(* IEC 61131-3 sources: ConveyorControl-with-PLC/4E_Gruppe1_Graf_Projekt1/Class/SdiasManager (part 3) *)

//**********************************************************************************************************************************************************
    CMD_GET_HARDWARE_DIAGNOSIS:
      //Returns module info
      ret_code := ERROR;
      pResult^.aData[0]$t_HWCGetHardwareDiagnosisOut.retcode := _HWC_RETVAL_ERROR;

      pStr_HWTRequested := pPara^.aPara[0]$t_HWCGetHardwareDiagnosisIn.pStr_HardewareTreeEntry;

      if pStr_HWTRequested &
         ( ((pStr_HWTRequested  + pPara^.aPara[0]$t_HWCGetHardwareTreeEntryIn.us_current_index  - 1)^$USINT) = HWT_ESCAPE_SDIAS ) then

        tmpplace := (pStr_HWTRequested+pPara^.aPara[0]$t_HWCGetHardwareDiagnosisIn.us_current_index)^$USINT;

        //Check if pointer is valid
        if ModuleObjInfo[tmpplace].pThis then
          ret_code := ModuleObjInfo[tmpplace].pThis^.NewInst(pPara,pResult);
        else
          pResult^.aData[0]$t_HWCGetHardwareDiagnosisOut.retcode := _HWC_RETVAL_ERROR_SDIAS_MODULE_NOT_FOUND;
        end_if;
      end_if;

//**********************************************************************************************************************************************************
    CMD_GET_HARDWARE_TREE_ENTRY:
      //Returns module info
      ret_code := ERROR;
      pResult^.aData[0]$t_HWCGetHardwareTreeEntryOut.retcode := _HWC_RETVAL_ERROR;

      pStr_HWTreeEntry := pPara^.aPara[0]$t_HWCGetHardwareTreeEntryIn.pStr_LastHardewareTreeEntry;

      //First HWT Path
      if pStr_HWTreeEntry = nil then
        if ModuleObjInfo[0].pThis then

          ret_code := ModuleObjInfo[0].pThis^.NewInst(pPara,pResult);
        else
          pResult^.aData[0]$t_HWCGetHardwareTreeEntryOut.retcode := _HWC_RETVAL_ERROR_SDIAS_MODULE_NOT_FOUND;
        end_if;

      //search next module
      elsif ( ((pStr_HWTreeEntry  + pPara^.aPara[0]$t_HWCGetHardwareTreeEntryIn.us_current_index  - 1)^$USINT) = HWT_ESCAPE_SDIAS ) then

        // Check last modul again incase it was an extension module
        usNextPlace := (pStr_HWTreeEntry  + pPara^.aPara[0]$t_HWCGetHardwareTreeEntryIn.us_current_index)^$USINT;
        if ModuleObjInfo[usNextPlace].pThis then

          ret_code := ModuleObjInfo[usNextPlace].pThis^.NewInst(pPara,pResult);
        else
          ret_code := READY;
          pResult^.aData$t_HWCGetHardwareTreeEntryOut.retcode := _HWC_RETVAL_OK_END_OF_LIST;
          return;
        end_if;

        // Module was found, return next one
        if ret_code = READY &
           (pResult^.aData$t_HWCGetHardwareTreeEntryOut.retcode = _HWC_RETVAL_OK_MODULE_FOUND |
            pResult^.aData$t_HWCGetHardwareTreeEntryOut.retcode = _HWC_RETVAL_OK_END_OF_LIST) then

          usNextPlace += 1;
          if ModuleObjInfo[usNextPlace].pThis then

            ret_code := ModuleObjInfo[usNextPlace].pThis^.NewInst(pPara,pResult);
          else
            ret_code := READY;
            pResult^.aData$t_HWCGetHardwareTreeEntryOut.retcode := _HWC_RETVAL_OK_END_OF_LIST;
          end_if;

        end_if;

      end_if;

//**********************************************************************************************************************************************************

//*****************************************************************************
//** COMMANDS FROM SDIAS MODULES                                             **
//*****************************************************************************

    // port number is always stored in pPara^.aPara[MAXCMDPARA-1]
//**********************************************************************************************************************************************************
		SDIAS_CMD_ADD_RD_ACCESS:
      if AddAccess(_Read, pPara^.aPara[0]$^SdiasBase, pPara^.aPara[1]$UDINT, pPara^.aPara[2], pPara^.aPara[3]$HINT, pPara^.aPara[4]$UINT, pPara^.aPara[5]$pVoid, pPara^.aPara[6]$pVoid, pPara^.aPara[7]$pVoid, pPara^.aPara[8]$^UDINT, pPara^.aPara[9]$UDINT, pPara^.aPara[10]$BOOL) = FALSE then
        ret_code := ERROR;
      end_if;

//**********************************************************************************************************************************************************
    SDIAS_CMD_ADD_WR_ACCESS:
      if AddAccess(_Write, pPara^.aPara[0]$^SdiasBase, pPara^.aPara[1]$UDINT, pPara^.aPara[2], pPara^.aPara[3]$HINT, pPara^.aPara[4]$UINT, pPara^.aPara[5]$pVoid, pPara^.aPara[6]$pVoid, pPara^.aPara[7]$pVoid, pPara^.aPara[8]$^UDINT, pPara^.aPara[9]$UDINT, pPara^.aPara[10]$BOOL) = FALSE then
        ret_code := ERROR;
      end_if;

//**********************************************************************************************************************************************************
		SDIAS_CMD_ADD_DYN_RD_ACCESS:
      if AddAccess(_ReadDynamic, pPara^.aPara[0]$^SdiasBase, pPara^.aPara[1]$UDINT, pPara^.aPara[2], pPara^.aPara[3]$HINT, pPara^.aPara[4]$UINT, pPara^.aPara[5]$pVoid, pPara^.aPara[6]$pVoid, pPara^.aPara[7]$pVoid, pPara^.aPara[8]$^UDINT, pPara^.aPara[9]$UDINT, pPara^.aPara[10]$BOOL) = FALSE then
        ret_code := ERROR;
      end_if;

//**********************************************************************************************************************************************************
    SDIAS_CMD_ADD_DYN_WR_ACCESS:
      if AddAccess(_WriteDynamic, pPara^.aPara[0]$^SdiasBase, pPara^.aPara[1]$UDINT, pPara^.aPara[2], pPara^.aPara[3]$HINT, pPara^.aPara[4]$UINT, pPara^.aPara[5]$pVoid, pPara^.aPara[6]$pVoid, pPara^.aPara[7]$pVoid, pPara^.aPara[8]$^UDINT, pPara^.aPara[9]$UDINT, pPara^.aPara[10]$BOOL) = FALSE then
        ret_code := ERROR;
      end_if;

//**********************************************************************************************************************************************************
    SDIAS_CMD_CHANGE_DYN_ACCESS:
      if ChangeDynAccess(AccessHandle:=pPara^.aPara[0]$UDINT, NewOffset:=pPara^.aPara[1]$UDINT, NewLength:=pPara^.aPara[2]$UDINT) = FALSE then
        ret_code := ERROR;
      end_if;

//**********************************************************************************************************************************************************
    SDIAS_CMD_SDO_SEND_REQUEST:

      if pPara^.aPara[1]$t_SDIAS_SDO_Cmd = SDIAS_SDO_CMD_SPI_READ & FirmwareVersion < SDIAS_SDO_SPI_FIRMWARE_VERSION_AVAILABLE then
        LogError(e_msg:="SdiasManager::ClassState::NewInst: SPI Read failed, Update FirmwareVersion of SDIAS Manager");
        ret_code := ERROR;
        return;
      end_if;

      if AddSDOReq(pCmdSvr:=pPara^.aPara[0]$^SvrChCmd, Command:=pPara^.aPara[1]$t_SDIAS_SDO_Cmd, Place:=pPara^.aPara[2]$USINT, CmdLength:=pPara^.aPara[3]$USINT, pReqBuf:=pPara^.aPara[4]$^USINT) <> SDIAS_OK then
        ret_code := ERROR;
      end_if;

//**********************************************************************************************************************************************************
    SDIAS_CMD_CHANGE_LED_STATE:
      // get byte position ouf of place (place 0-3 in byte 0, 4-7 in byte 1,...)
      ByteNr := pPara^.aPara[1]$USINT SHR 2;
      PosInByte := (pPara^.aPara[1]$USINT AND 2#11) SHL 1;
      AppliLEDStates[ByteNr] := (AppliLEDStates[ByteNr] AND NOT(2#11 SHL PosInByte)) OR (pPara^.aPara[2]$USINT SHL PosInByte);
      b_NewLEDStates := TRUE;

//**********************************************************************************************************************************************************
    SDIAS_CMD_DA_RD_ACCESS:
      // not implemented yet
      ret_code := ERROR;

//      DaWriteBuffer.ReadLength  := pPara^.aPara[1]$USINT;
//      DaWriteBuffer.ReadOffset  := pPara^.aPara[0]$HINT;
//      DaWriteBuffer.WriteLength := 0;
//      DaWriteBuffer.WriteOffset := 0;
//
//      DaWriteBuffer.TriggerUnit := sizeof(t_DAWrPayloadFrame) - sizeof(t_DAWrPayloadFrame.Data); // no data sent on reading
//
//      DAPara.ud_AddOffset := DaWriteOffset;
//      DAPara.ud_length    := DaWriteBuffer.TriggerUnit;
//      DAPara.p_ud_data    := (#DaWriteBuffer)$^UDINT;
//
//      tempCmd.uiCmd := _BUS_IF_WR_DA;
//      tempCmd.aPara[0] := (#DAPara)$DINT;
//      ToBusInterface.NewInst(pPara:=#tempCmd, pResult:=#_result);
//
//      if _result.aData[4]$t_BusIFRetvalErrorcode <> _BUS_IF_RETVAL_OK then
//        LogError("(SdiasManager::ClassState::NewInst) Direct access write on VARAN failed as part of the SDIAS direct access read!");
//        ret_code := ERROR;
//      else
//        DAPara.ud_AddOffset := DaReadOffset;
//        DAPara.ud_length    := DaWriteBuffer.ReadLength + sizeof(t_SDIAS_StateByte);
//        DAPara.p_ud_data    := (#DaReadBuffer)$^UDINT;
//
//        tempCmd.uiCmd := _BUS_IF_RD_DA;
//        tempCmd.aPara[0] := (#DAPara)$DINT;
//        ToBusInterface.NewInst(pPara:=#tempCmd, pResult:=#_result);
//
//        if _result.aData[4]$t_BusIFRetvalErrorcode <> _BUS_IF_RETVAL_OK then
//          LogError("(SdiasManager::ClassState::NewInst) Direct access read on VARAN failed as part of the SDIAS direct access read!");
//          ret_code := ERROR;
//        else
//          // copy the read data to the user memory
//          _memcpy(ptr1:=pPara^.aPara[2]$^USINT, ptr2:=#DaReadBuffer.Data, cntr:=DaWriteBuffer.ReadLength);
//        end_if;
//      end_if;

//**********************************************************************************************************************************************************
    SDIAS_CMD_DA_WR_ACCESS:
      // not implemented yet
      ret_code := ERROR;

//      DaWriteBuffer.ReadLength  := 0;
//      DaWriteBuffer.ReadOffset  := 0;
//      DaWriteBuffer.WriteLength := pPara^.aPara[1]$USINT;
//      DaWriteBuffer.WriteOffset := pPara^.aPara[0]$HINT;
//
//      DaWriteBuffer.TriggerUnit := sizeof(t_DAWrPayloadFrame) - sizeof(t_DAWrPayloadFrame.Data) + DaWriteBuffer.WriteLength; // no data sent on reading
//
//      // copy the write data from the user memory
//      _memcpy(ptr1:=#DaWriteBuffer.Data, ptr2:=pPara^.aPara[2]$^USINT, cntr:=DaWriteBuffer.WriteLength);
//
//      DAPara.ud_AddOffset := DaWriteOffset;
//      DAPara.ud_length    := DaWriteBuffer.TriggerUnit;
//      DAPara.p_ud_data    := (#DaWriteBuffer)$^UDINT;
//
//      tempCmd.uiCmd := _BUS_IF_WR_DA;
//      tempCmd.aPara[0] := (#DAPara)$DINT;
//      ToBusInterface.NewInst(pPara:=#tempCmd, pResult:=#_result);
//
//      if _result.aData[4]$t_BusIFRetvalErrorcode <> _BUS_IF_RETVAL_OK then
//        LogError("(SdiasManager::ClassState::NewInst) Direct access write on VARAN failed as part of the SDIAS direct access write!");
//        ret_code := ERROR;
//      else
//        DAPara.ud_AddOffset := DaReadOffset;
//        DAPara.ud_length    := sizeof(t_SDIAS_StateByte);
//        DAPara.p_ud_data    := (#DaReadBuffer)$^UDINT;
//
//        tempCmd.uiCmd := _BUS_IF_RD_DA;
//        tempCmd.aPara[0] := (#DAPara)$DINT;
//        ToBusInterface.NewInst(pPara:=#tempCmd, pResult:=#_result);
//
//        if _result.aData[4]$t_BusIFRetvalErrorcode <> _BUS_IF_RETVAL_OK then
//          LogError("(SdiasManager::ClassState::NewInst) Direct access read on VARAN failed as part of the SDIAS direct access write!");
//          ret_code := ERROR;
//        end_if;
//      end_if;

//**********************************************************************************************************************************************************
    SDIAS_CMD_REQUIRED_ERROR:
      SetRequiredError(pTargetThis:=pPara^.aPara[0]$^SdiasBase, Place:=pPara^.aPara[1]$UDINT);

//**********************************************************************************************************************************************************
    SDIAS_CMD_INIT_STATE_LOGIN:
      Place := pPara^.aPara[1]$UDINT;
      if (Place <= SDIAS_MAX_PLACE_NR) & pPara^.aPara[0] then
        ModuleObjInfo[Place].pInitState       := pPara^.aPara[0]$^t_e_VaranErrors;
        ModuleObjInfo[Place].pThis            := pPara^.aPara[2]$^SdiasBase;

        // get task settings
        ModuleObjInfo[Place].bPreScan         := (pPara^.aPara[3] AND SDIAS_TASK_MASK_RT_PRE ) <> 0;
        ModuleObjInfo[Place].bPostScan        := (pPara^.aPara[3] AND SDIAS_TASK_MASK_RT_POST) <> 0;
        ModuleObjInfo[Place].bCyclic          := (pPara^.aPara[3] AND SDIAS_TASK_MASK_CY     ) <> 0;

        // get access structure
        ModuleObjInfo[Place].pDefaultAccesses := pPara^.aPara[4]$^t_SDIAS_DefaultAccesses;

        // required info
        ModuleObjInfo[Place].Required         := pPara^.aPara[5];

        if ModuleObjInfo[Place].Required & (b_SDIASModulesRequired = FALSE) then
          b_SDIASModulesRequired := TRUE;
          // if any access is required => the businterface is also required
          tempCmd.uiCmd := _BUS_IF_SET_REQUIRED;
          ToBusInterface.NewInst(pPara:=#tempCmd, pResult:=#_result);
          if _result.aData[0]$t_BusIFRetvalErrorcode <> _BUS_IF_RETVAL_OK then
            LogError("(SdiasManager::ClassState::NewInst) Failed to set the BusInterface to required");
          end_if;
        end_if;

        // remember the highest place to save time in module scanning operations like calling the realtime methods
        if (Place > MaxPlace) | (MaxPlace = SDIAS_PLACE_NO_MODULE_ADDED_SO_FAR) then
          MaxPlace := Place;
        end_if;
      else
        ret_code := ERROR;
      end_if;

//**********************************************************************************************************************************************************
    SDIAS_CMD_GET_HW_PATH:
      // forward it to bus interface
      pPara^.uiCmd := _BUS_IF_GET_HW_PATH;
      ret_code := ToBusInterface.NewInst(pPara, pResult);

//**********************************************************************************************************************************************************
    SDIAS_CMD_INSTALL_CYCLIC_TASK:
      ModuleObjInfo[pPara^.aPara[0]].bCyclic := TRUE;

//**********************************************************************************************************************************************************
    SDIAS_CMD_GET_CONNECTION_TYPE:
      pResult^.uiLng := sizeof(t_SDIAS_ConnectionType);
      pResult^.aData[0]$t_SDIAS_ConnectionType := ConnectionType;

//**********************************************************************************************************************************************************
    SDIAS_CMD_CREATE_MUTEX:
      // forward it to bus interface
      pPara^.uiCmd := _BUS_IF_CREATE_MUTEX;
      ret_code := ToBusInterface.NewInst(pPara, pResult);

//**********************************************************************************************************************************************************
    SDIAS_CMD_IS_VARAN_AVAILABLE:
      // forward it to bus interface
      pPara^.uiCmd := _BUS_IF_IS_VARAN_AVAILABLE;
      ret_code := ToBusInterface.NewInst(pPara, pResult);

//**********************************************************************************************************************************************************
    SDIAS_CMD_ADD_DEVICE_ID:
    //add valid ids to list
    for i:= 0 to 9 do
      //Check if no id is stored or if id is already stored in list.
      if aValidDeviceIDs[i] = 0 | aValidDeviceIDs[i] = pPara^.aPara[0]$UDINT then
        aValidDeviceIDs[i] := pPara^.aPara[0]$UDINT;
        exit;
      end_if;
    end_for;

//**********************************************************************************************************************************************************

//*****************************************************************************
//** COMMANDS FORWARDED BY SDIAS BUS INTERFACE                               **
//*****************************************************************************

//**********************************************************************************************************************************************************
    _BUS_IF_ADD_MOVE_DO:
      // correct the parameters, because the calling class doesn't have the information
      pDataADDMove                        := (pPara^.aPara[0])$^t_AddMoveDOCfg;

      pDataADDMove^.ud_handle_source      := ISOReadDO.AccessHandle;
      pDataADDMove^.ud_addressoff_source  := pDataADDMove^.p_sourcedata$UDINT - ISOReadDO.pData$UDINT;

      // if we have the DPRAM address extra => recalculate the address
      if ISOReadDO.pDataDPRAM then
        pDataADDMove^.p_sourcedata := ISOReadDO.pDataDPRAM + pDataADDMove^.ud_addressoff_source;
      end_if;

      pDataADDMove^.ud_handle_dest        := ISOWriteDO.AccessHandle;
      pDataADDMove^.ud_addressoff_dest    := pDataADDMove^.p_destdata$UDINT - ISOWriteDO.pData$UDINT;

      // if we have the DPRAM address extra => recalculate the address
      if ISOWriteDO.pDataDPRAM then
        pDataADDMove^.p_destdata := ISOWriteDO.pDataDPRAM + pDataADDMove^.ud_addressoff_dest;
      end_if;

      // forward it to bus interface
      ret_code := ToBusInterface.NewInst(pPara, pResult);

//**********************************************************************************************************************************************************
    _BUS_IF_UPDATE_MOVE_DO:
      // forward it to bus interface
      ret_code := ToBusInterface.NewInst(pPara, pResult);

//**********************************************************************************************************************************************************
    _BUS_IF_GET_ACCESS_INFO:
      // check if we got a valid pointer (local memory)
      if pPara^.aPara[0] then
        // return the access info
        pResult^.uiLng := sizeof(t_AccessInfoRet);
        pAccessInfo := (#pResult^.aData[0])$^t_AccessInfoRet;

        pAccessInfo^.ud_handle     := ISOReadDO.AccessHandle;
        pAccessInfo^.ud_addressoff := pPara^.aPara[0]$UDINT - ISOReadDO.pData$UDINT;

        // if we have the DPRAM address extra => recalculate the address
        if ISOReadDO.pDataDPRAM then
          pAccessInfo^.p_dataDPRAM := ISOReadDO.pDataDPRAM + pAccessInfo^.ud_addressoff;
        end_if;
      end_if;

//**********************************************************************************************************************************************************

//*****************************************************************************
//** COMMANDS FROM BUS INTERFACE                                             **
//*****************************************************************************

//**********************************************************************************************************************************************************
    _BUS_IF_HWCONNECT :
      // device has been connected. if there is no bus ready signal or we're in the init (no bus ready in init if module is already connected) => do the connect-stuff here
      ConnectEvent();
      pResult^.aData[0] := _BUS_IF_RETVAL_OK;

//**********************************************************************************************************************************************************
    _BUS_IF_HWSUB_BUS_READY :
      // we wait for the device bitmap to match => do nothing here
      pResult^.aData[0] := _BUS_IF_RETVAL_OK;

//**********************************************************************************************************************************************************
    _BUS_IF_HWDISCONNECT :
      // device has been disconnected
      DisconnectEvent();
      pResult^.aData[0] := _BUS_IF_RETVAL_OK;

//**********************************************************************************************************************************************************
    _BUS_IF_HWINTERRUPT :
      // error at device which may lead to a disconnect or replace the disconnect callback
      InterruptEvent();
      pResult^.aData[0] := _BUS_IF_RETVAL_OK;

//**********************************************************************************************************************************************************
    _BUS_IF_CHECK_DEVICE_ID :
      // check for correct device id

      pResult^.aData[0] := (DeviceID = pPara^.aPara[0]$UDINT);
      if pResult^.aData[0] = false then
        for i:= 0 to 9 do
          //Id found?
          if aValidDeviceIDs[i] = pPara^.aPara[0]$UDINT then
            pResult^.aData[0] := TRUE;
            exit;
          end_if;
        end_for;
      end_if;

//**********************************************************************************************************************************************************
    _BUS_IF_GET_TASK_INFO:
      // we must fetch the task info before the image with the payload is copied to ensure correct data and correct error detection

      // on local SDIAS we have to fetch it from the OS
      if ConnectionType = SDIAS_CON_LOCAL_uC then
        if SDIAS_iGetNodePropertyIndexLen(hNodeHandle   := udNodeHandle
                                     , udIndex          := 1
                                     , udPropertyId     := SDM_PROP_TASK_INFO
                                     , udBufferLength   := sizeof(t_TaskInfoData) - sizeof(t_TaskInfoData.ErrorInfoFlags) - sizeof(t_TaskInfoData.Reserved)
                                     , pucBuf           := (#RdTaskInfo.Handshake)$^USINT
                                     ) <> SDIAS_OK then
          CyclicMsgMarker.PostIt.GetRdInfoFailed := TRUE;
        end_if;
        if SDIAS_iGetNodePropertyIndex(hNodeHandle      := udNodeHandle
                                     , udIndex          := 1
                                     , udPropertyId     := SDM_PROP_TASK_ERROR_INFO_FLAGS
                                     , pudPropertyValue := (#RdTaskInfo.ErrorInfoFlags)$^UDINT
                                     ) <> SDIAS_OK then
          CyclicMsgMarker.PostIt.GetRdInfoFailed := TRUE;
        end_if;

        if SDIAS_iGetNodePropertyIndexLen(hNodeHandle   := udNodeHandle
                                     , udIndex          := 2
                                     , udPropertyId     := SDM_PROP_TASK_INFO
                                     , udBufferLength   := sizeof(t_TaskInfoData) - sizeof(t_TaskInfoData.ErrorInfoFlags) - sizeof(t_TaskInfoData.Reserved)
                                     , pucBuf           := (#WrTaskInfo.Handshake)$^USINT
                                     ) <> SDIAS_OK then
          CyclicMsgMarker.PostIt.GetWrInfoFailed := TRUE;

        end_if;
        if SDIAS_iGetNodePropertyIndex(hNodeHandle      := udNodeHandle
                                     , udIndex          := 2
                                     , udPropertyId     := SDM_PROP_TASK_ERROR_INFO_FLAGS
                                     , pudPropertyValue := (#WrTaskInfo.ErrorInfoFlags)$^UDINT
                                     ) <> SDIAS_OK then
          CyclicMsgMarker.PostIt.GetWrInfoFailed := TRUE;
        end_if;
      end_if;

//**********************************************************************************************************************************************************
    _BUS_IF_POST_INIT_RT_READY:
      // if we got an error => return it
      if InitSSW = _ErrorOccured then
        ret_code := ERROR;

      // if we're not ready, return busy
      elsif RtSSW <> _Operational then
        ret_code := BUSY;
      end_if;

//**********************************************************************************************************************************************************
    _BUS_IF_CREATE_MUTEX,
    _BUS_IF_SET_REQUIRED_ERROR,
    _BUS_IF_GET_BUSCYCLE_TIME,
    _BUS_IF_GET_DEACTIVATED_STATE,
    _BUS_IF_GET_HW_PATH,
    _BUS_IF_IS_VARAN_AVAILABLE,
    _BUS_IF_SET_RUN_STATE,
    _BUS_IF_SET_REQUIRED:
      // forward it to bus interface
      ret_code := ToBusInterface.NewInst(pPara, pResult);
//**********************************************************************************************************************************************************

//*****************************************************************************
//** COMMANDS FROM SDIAS MANAGER ITSELF                                      **
//*****************************************************************************

//**********************************************************************************************************************************************************
		SDIAS_CMD_SDO_RESPONSE:
      ret_code := ReceiveSDOResponse(Command:=pPara^.aPara[0]$t_SDIAS_SDO_Cmd,
                                     Offset:=pPara^.aPara[1]$HINT,
                                     Length:=pPara^.aPara[2]$USINT,
                                     Result:=pPara^.aPara[3]$iprStates,
                                     pResponseBuffer:=pPara^.aPara[4]$^USINT,
                                     ResponseLength:=pPara^.aPara[5]$USINT
                                     );

//**********************************************************************************************************************************************************
  else
    // unknown command
    LogValue("(SdiasManager::ClassState::NewInst) Unknown command: 0x{0}", pPara^.uiCmd);
    ret_code := ERROR;
	END_CASE;

END_FUNCTION

FUNCTION SdiasManager::AddAccess
	VAR_INPUT
		AccessType 	: t_eAccessType;
		pThis 	: ^SdiasBase;
		Place 	: UDINT;
		Required 	: DINT;
		Offset 	: HINT;
		Length 	: UINT;
		ppData 	: pVoid;
		ppStateByte 	: pVoid;
		ppControlByte 	: pVoid;
		pAccessHandle 	: ^UDINT;
		WaitForAccessHandle 	: UDINT;
		bCtrlAcc0 	: BOOL;
	END_VAR
	VAR_OUTPUT
		Success 	: BOOL;
	END_VAR

  // check place
  if Place <= SDIAS_MAX_PLACE_NR then
    // check this pointer
    if pThis then
      // check other pointers as input parameters
      if ppData & ppStateByte & ppControlByte then
        // check offset and length for valid access
        if (Length > 0) & ((Offset + Length) <= SIZE_PER_SDIAS_CLIENT) then

          // remember the highest place to save time in module scanning operations like calling the realtime methods
          if (Place > MaxPlace) | (MaxPlace = SDIAS_PLACE_NO_MODULE_ADDED_SO_FAR) then
            MaxPlace := Place;
          end_if;

          // if it's a dynamic access on local SDIAS, check if the OS-Interface is available
          if ConnectionType = SDIAS_CON_LOCAL_uC then
            if ((AccessType = _ReadDynamic) | (AccessType = _WriteDynamic)) & (pSDIAS^.udVersion < SDIAS_CIL_VERSION_SUPPORTS_DYNAMIC_DO) then
              LogValue("(SdiasManager::AddAccess) Newer OS Version needed for dynamic accesses on local SDIAS. Access for module at place 0x{0} can't be created!", Place);
              ModuleObjInfo[Place].pInitState^ := _UnknownCommand;
              InitError := _UnknownCommand;
              Success := FALSE;
              return;
            end_if;
          end_if;

          // remember the access
          Success := AddAccessToList(AccessType           := AccessType,
                                     Place                := Place,
                                     Offset               := Offset,
                                     Length               := Length,
                                     ppData               := ppData,
                                     ppStateByte          := ppStateByte,
                                     ppControlByte        := ppControlByte,
                                     pAccessHandle        := pAccessHandle,
                                     WaitForAccessHandle  := WaitForAccessHandle,
                                     bCtrlAcc0            := bCtrlAcc0
                                     );

          // if adding failed classstate and initerrorstate are already set
          if Success = FALSE then
            LogValue("(SdiasManager::AddAccess) Failed to add Access for Module at Place 0x{0}", Place);
          end_if;
        else
          LogValue("(SdiasManager::AddAccess) Invalid access for module at place: 0x{0}. Check offset (0x{1}) and length (0x{2})!", Place, Offset, Length);
          ModuleObjInfo[Place].pInitState^ := _DOLAddressInvalid;
          InitError := _DOLAddressInvalid;
          Success := FALSE;
        end_if;
      else
        LogValue("(SdiasManager::AddAccess) Invalid pointer as input parameter for module at place: 0x{0}", Place);
        ModuleObjInfo[Place].pInitState^ := _MemoryFault;
        InitError := _MemoryFault;
        Success := FALSE;
      end_if;
    else
      LogValue("(SdiasManager::AddAccess) Invalid this pointer for module at place: 0x{0}", Place);
      ModuleObjInfo[Place].pInitState^ := _MemoryFault;
      InitError := _MemoryFault;
      Success := FALSE;
    end_if;
  else
    LogValue("(SdiasManager::AddAccess) Invalid Place number: 0x{0}. Maximum is 0x{1}", Place, SDIAS_MAX_PLACE_NR);
    if pThis then
      pThis^.ClassState := _InvalidDeviceAddress;
    end_if;
    InitError := _InvalidDeviceAddress;
    Success := FALSE;
  end_if;

  // if it was an access of a required module => required error
  if Required & (Success = FALSE) then
    SetRequiredError(pThis, Place);
  end_if;

END_FUNCTION

FUNCTION SdiasManager::ConnectEvent
  VAR
  	tempCmd         : CmdStruct;
    _result         : results;
    dataResetDO     : t_ResetDOCfg;
    Settings        : t_LoginSettings;
  END_VAR

  if b_PostInitFinished = FALSE then
    ConnectDuringPostInitCounter += 1;

    // don't reinit in postinit (ignore call from OS)
    if ConnectDuringPostInitCounter >= 2 then
      b_MultipleConnectInInit := TRUE;
      return;
    end_if;
  end_if;

  // install post init call back only if we're still in init (if we install it in init(), we may get called even the module is not connected)
  if us_Firstscan < 12 then
    tempCmd.uiCmd := _BUS_IF_WAIT_4_POST_INIT;
#pragma warning(disable: 74);
    Settings := 0;
#pragma warning(default: 74);
    Settings.Wait4DOCreation := MaxPlace <> SDIAS_PLACE_NO_MODULE_ADDED_SO_FAR;
    if Settings.Wait4DOCreation & (ConnectionType = SDIAS_CON_VIA_VARAN_uC) then
      Settings.Wait4MoveDOCreation := TRUE;
    end_if;
    Settings.Wait4SyncSend := TRUE;

    tempCmd.aPara[0] := Settings;
    ToBusInterface.NewInst(pPara:=#tempCmd, pResult:=#_result);

    if _result.aData[0]$t_BusIFRetvalErrorcode <> _BUS_IF_RETVAL_OK then
      LogError("(SdiasManager::ClassState::NewInst) Failed to install post init callback");
      InitError := _InvalidConfguration;
    end_if;
  else
    b_PostInitFinished := TRUE;
  end_if;

  if ConnectionType = SDIAS_CON_VIA_VARAN_uC then

    // reset data objects (calculate retry timeout)
    tempCmd.uiCmd     := _BUS_IF_RESET_DO;
    tempCmd.aPara[0]  := (#dataResetDO)$DINT;

    dataResetDO.Handle := ASYReadDO.Handle;

    ToBusInterface.NewInst(pPara:=#tempCmd, pResult:=#_result);
    if _result.aData[0]$t_BusIFRetvalErrorcode <> _BUS_IF_RETVAL_OK then
      LogError("(SdiasManager::ConnectEvent) Failed reset DO for the asynchronous read data");
    end_if;

    dataResetDO.Handle := ASYWriteDO.Handle;

    ToBusInterface.NewInst(pPara:=#tempCmd, pResult:=#_result);
    if _result.aData[0]$t_BusIFRetvalErrorcode <> _BUS_IF_RETVAL_OK then
      LogError("(SdiasManager::ConnectEvent) Failed reset DO for the asynchronous write data");
    end_if;
  end_if;

  // reset max durations as it marks the first run
  WriteTaskInfo.MaxDuration := 0;
  ReadTaskInfo.MaxDuration := 0;

  InitSSW := _StartInit;
  b_Ready4Rt := FALSE;
  RtSSW := _RtIdle;
  ClassState := _NotInitialized;
  Online := 1;

END_FUNCTION

FUNCTION SdiasManager::DisconnectEvent
  VAR
  	i : UDINT;
  END_VAR

  // if there is a required error, we would disguise it, if we call the disconnect interfaces
  if ClassState <> _RequiredError then

    // tell all the connected modules
    if MaxPlace <> SDIAS_PLACE_NO_MODULE_ADDED_SO_FAR then
      for i := 0 to MaxPlace do
        if ModuleObjInfo[i].pThis then
          ModuleObjInfo[i].pThis^.DisconnectEvent();
        end_if;
      end_for;
    end_if;

    ClassState := _NoHardware;

    FirmwareVersion := 0;
  end_if;

  Online := 0;

END_FUNCTION

FUNCTION SdiasManager::InterruptEvent

  // set only the state (we're in the interrupt and have to be fast)
  if b_IsRequired then
    ClassState := _HardwareRequiredIRQ;
  else
    ClassState := _HardwareNotRequiredIRQ;
  end_if;

  Online := 0;

END_FUNCTION

FUNCTION SdiasManager::SdiasManager
	VAR_OUTPUT
		ret_code 	: ConfStates;
	END_VAR
  VAR
    p_SSR			: ^LSL_SSR;
  END_VAR

  ClassState := _NotInitialized;

  //get pointer for logging function
	if ( OS_CILGET( "SSR", #p_SSR ) ) then
    p_KernelLog := NIL;
  else
    //Log function is available
		p_KernelLog := ( p_SSR^.KernelLog )$^DINT;
  end_if;

  //get pointer for sdias function
	if OS_CILGET( INTERFACE_SDIAS, #pSDIAS ) then
    LogError(e_msg:="(SdiasManager::SdiasManager) Failed to get SDIAS OS-Interface. A newer OS is necessary to use SDIAS");
  end_if;

  if (OS_CILGet("LSL_MULTITASK", #mt_api$void)) THEN
    LogError(e_msg:="(SdiasManager::SdiasManager) Failed to get MULTITASK OS-Interface for Mutex usage");
  end_if;

  MaxPlace := SDIAS_PLACE_NO_MODULE_ADDED_SO_FAR;

	ret_code := C_OK;

END_FUNCTION

FUNCTION VIRTUAL SdiasManager::LogError
	VAR_INPUT
		e_msg 	: ^CHAR;
	END_VAR
  VAR
    sz_name : ARRAY [ 0..255 ] OF CHAR;
  END_VAR

  _GetObjName( this, #sz_name[ 0 ] );

  MyTrace(pFormat:="ObjectName {0}: {1}", pTxt0:=(#sz_name[ 0 ])$^CHAR, pTxt1:= e_msg, pTxt2:=NIL);

END_FUNCTION

FUNCTION VIRTUAL SdiasManager::LogValue
	VAR_INPUT
		pString 	: ^CHAR;
		Value 	: UDINT;
		Value2 	: UDINT;(* := 16#FFFFFFFF *)
		Value3 	: UDINT;(* := 16#FFFFFFFF *)
	END_VAR
  VAR
    TempStr       : ARRAY [0..99] OF CHAR;
    TempStr2      : ARRAY [0..99] OF CHAR;
    TempStr3      : ARRAY [0..99] OF CHAR;
    TraceVal      : USINT;
    sz_name       : ARRAY [ 0..255 ] OF CHAR;
    TmpWithObjName: ARRAY [ 0..255 ] OF CHAR;
  END_VAR

  // number of values
  TraceVal := 1;

  _itoa(Value, #TempStr[0]);

  if pString <> NIL then
    _GetObjName( this, #sz_name[ 0 ] );
    _strcpy(dest:=#TmpWithObjName[0], src:="ObjectName ");
    _strcat(dest:=#TmpWithObjName[0], src:=#sz_name[0]);
    _strcat(dest:=#TmpWithObjName[0], src:=": ");
    _strcat(dest:=#TmpWithObjName[0], src:=pString);

    if Value2 <> 16#FFFFFFFF then
      _itoa(Value2, #TempStr2[0]);
      TraceVal += 1;
    end_if;

    if Value3 <> 16#FFFFFFFF then
      _itoa(Value3, #TempStr3[0]);
      TraceVal += 1;
    end_if;

    case TraceVal of
      1:MyTrace(pFormat:=#TmpWithObjName[0], pTxt0:=#TempStr[0], pTxt1:=NIL, pTxt2:=NIL);
      2:MyTrace(pFormat:=#TmpWithObjName[0], pTxt0:=#TempStr[0], pTxt1:=#TempStr2[0], pTxt2:=NIL);
      3:MyTrace(pFormat:=#TmpWithObjName[0], pTxt0:=#TempStr[0], pTxt1:=#TempStr2[0], pTxt2:=#TempStr3[0]);
    end_case;
  else
    MyTrace(pFormat:="<invalid string>", pTxt0:=NIL, pTxt1:=NIL, pTxt2:=NIL);
  end_if;

END_FUNCTION

FUNCTION VIRTUAL SdiasManager::MyTrace
	VAR_INPUT
		pFormat 	: ^CHAR;
		pTxt0 	: ^CHAR;
		pTxt1 	: ^CHAR;
		pTxt2 	: ^CHAR;
	END_VAR
  VAR
    nLen      : UDINT;
    pChr      : ^CHAR;
    nTxt      : UDINT;
    nRpl      : UDINT;
    pTxt      : ^CHAR;
    pText     : ^CHAR;
    FormText  : ARRAY [0 .. 255] OF CHAR;
  END_VAR

  // this method is a workaround for the TRACE message limitation problem

  pText := #FormText[0];

  _memset(dest:=#FormText[0], usByte:=0, cntr:=256); // to keep the zero termination

  _strncpy(pText, pFormat, 250);
  nLen  := _strlen(pText);
  pChr  := pText;

  WHILE nLen DO
    IF pChr^ = '{' THEN         // works for the first 10 replacement texts (single digit numbers)
      nTxt  := (pChr+1)^ - '0';
      CASE nTxt OF
        0:  pTxt  := pTxt0;
        1:  pTxt  := pTxt1;
        2:  pTxt  := pTxt2;
      ELSE
        pTxt  := "INV";
      END_CASE;
      nRpl  := _strlen(pTxt);
      if nLen - 3 + nRpl > 250 then
        pTxt := "LEN";  // replace the replacement text with "LEN" to see that we're out of length for this string
        nRpl := 3;
      end_if;
      _memmove(pChr + nRpl, pChr + 3, nLen);
      _memcpy(pChr, pTxt, nRpl);
      pChr  += nRpl;  // next character to parse is after the replacement text
      nLen  -= 3;     // the remaining length of the format string is decremented by 3
      if nLen > 250 then  // catch overrun of nLen
        nLen := 0;
      end_if;
    ELSE
      pChr  += 1;
      nLen  -= 1;
    END_IF;
  END_WHILE;

  TRACE(#FormText[0]);
  if ( p_KernelLog ) then
    OS_KERNELLOG0(#FormText[0]);
  end_if;

END_FUNCTION

FUNCTION SdiasManager::ChangeAsyRd
	VAR_INPUT
		Offset 	: HINT;
		Length 	: USINT;
		RunState 	: t_BusIFRunState;
		UsageType 	: t_AsyDOUsage;
	END_VAR
	VAR_OUTPUT
		Success 	: BOOL;
	END_VAR
  VAR
    dataUPDATEDO    : t_UpdateDOCfg;
  	tempCmd         : CmdStruct;
    _result         : results;
    dataSETRUNSTATE : t_SetRunStateCfg;
  END_VAR

  if (AsyReadUsage = _NotUsed) | (AsyReadUsage = UsageType) then

    // if length = zero we may just want to stop the DO
    if Length then
      ASYReadDO.Offset := Offset;
      ASYReadDO.Length := Length;

      dataUPDATEDO.Handle               := ASYReadDO.Handle;
      dataUPDATEDO.ud_addressoff_read   := ASYReadDO.Offset;
      dataUPDATEDO.ud_length_read       := ASYReadDO.Length;

      tempCmd.uiCmd         := _BUS_IF_UPDATE_DO;
      tempCmd.aPara[0]      := (#dataUPDATEDO)$DINT;

      ToBusInterface.NewInst(pPara:=#tempCmd, pResult:=#_result);
      if _result.aData[0]$t_BusIFRetvalErrorcode <> _BUS_IF_RETVAL_OK then
        LogError("(SdiasManager::ChangeAsyRd) Failed to change asynchron read access");
      end_if;
    end_if;

    // set runstate
    dataSETRUNSTATE.Handle      := ASYReadDO.Handle;
    dataSETRUNSTATE.NewRunState := RunState;

    tempCmd.uiCmd         := _BUS_IF_SET_RUN_STATE;
    tempCmd.aPara[0]      := (#dataSETRUNSTATE)$DINT;

    ToBusInterface.NewInst(pPara:=#tempCmd, pResult:=#_result);

    if _result.aData[0]$t_BusIFRetvalErrorcode <> _BUS_IF_RETVAL_OK then
      LogError("(SdiasManager::ChangeAsyRd) Error changing the run state of the asynchron read access!");
    end_if;

    if RunState = _BUS_IF_RUN_STATE_NO_RUN then
      AsyReadUsage := _NotUsed;
    else
      AsyReadUsage := UsageType;
    end_if;

    Success := TRUE;
  else
    LogError("(SdiasManager::ChangeAsyRd) Failed to use DO (already in use by another task)");
    Success := FALSE;
  end_if;

END_FUNCTION

FUNCTION SdiasManager::ChangeAsyWr
	VAR_INPUT
		Offset 	: HINT;
		Length 	: USINT;
		RunState 	: t_BusIFRunState;
		UsageType 	: t_AsyDOUsage;
	END_VAR
	VAR_OUTPUT
		Success 	: BOOL;
	END_VAR
  VAR
    dataUPDATEDO    : t_UpdateDOCfg;
  	tempCmd         : CmdStruct;
    _result         : results;
    dataSETRUNSTATE : t_SetRunStateCfg;
  END_VAR

  if (AsyWriteUsage = _NotUsed) | (AsyWriteUsage = UsageType) then
    // if a watchdog trigger has to be sent, ignore other requests
    if b_SendWdTrigger & (UsageType <> _UsedByWD) then
      AsyWriteUsage := _UsedByWD;
      Success := FALSE;
      return;
    end_if;

    // if length = zero we may just want to stop the DO
    if Length then
      ASYWriteDO.Offset := Offset;
      ASYWriteDO.Length := Length;

      dataUPDATEDO.Handle               := ASYWriteDO.Handle;
      dataUPDATEDO.ud_addressoff_write  := ASYWriteDO.Offset;
      dataUPDATEDO.ud_length_write      := ASYWriteDO.Length;

      tempCmd.uiCmd         := _BUS_IF_UPDATE_DO;
      tempCmd.aPara[0]      := (#dataUPDATEDO)$DINT;

      ToBusInterface.NewInst(pPara:=#tempCmd, pResult:=#_result);
      if _result.aData[0]$t_BusIFRetvalErrorcode <> _BUS_IF_RETVAL_OK then
        LogError("(SdiasManager::ChangeAsyWr) Failed to change asynchron write access");
      end_if;
    end_if;

    // set runstate
    dataSETRUNSTATE.Handle      := ASYWriteDO.Handle;
    dataSETRUNSTATE.NewRunState := RunState;

    tempCmd.uiCmd         := _BUS_IF_SET_RUN_STATE;
    tempCmd.aPara[0]      := (#dataSETRUNSTATE)$DINT;

    ToBusInterface.NewInst(pPara:=#tempCmd, pResult:=#_result);

    if _result.aData[0]$t_BusIFRetvalErrorcode <> _BUS_IF_RETVAL_OK then
      LogError("(SdiasManager::ChangeAsyWr) Error changing the run state of the asynchron write access!");
    end_if;

    if RunState = _BUS_IF_RUN_STATE_NO_RUN then
      AsyWriteUsage := _NotUsed;
    else
      AsyWriteUsage := UsageType;
    end_if;

    Success := TRUE;
  else
    // only print the message if there is no collision with watchdog (collision with watchdog is very likely)
    if (AsyWriteUsage <> _UsedByWD) & (UsageType <> _UsedByWD) then
      LogError("(SdiasManager::ChangeAsyWr) Failed to use DO (already in use by another task)");
    end_if;

    Success := FALSE;
  end_if;

END_FUNCTION

FUNCTION SdiasManager::AddAccessToList
	VAR_INPUT
		AccessType 	: t_eAccessType;
		Place 	: UDINT;
		Offset 	: HINT;
		Length 	: UINT;
		ppData 	: pVoid;
		ppStateByte 	: pVoid;
		ppControlByte 	: pVoid;
		pAccessHandle 	: ^UDINT;
		WaitForAccessHandle 	: UDINT;
		bCtrlAcc0 	: BOOL;
	END_VAR
	VAR_OUTPUT
		Success 	: BOOL;
	END_VAR
  VAR
    pHelpAccess : ^t_AccessElement;
  END_VAR

  if ModuleObjInfo[Place].pFirstAccess = NIL then
    ModuleObjInfo[Place].pFirstAccess$pVoid := ToStdLib.Malloc(size:=sizeof(t_AccessElement));
    pHelpAccess := ModuleObjInfo[Place].pFirstAccess;
  else
    pHelpAccess := ModuleObjInfo[Place].pFirstAccess;
    while pHelpAccess^.pNext <> NIL do
      pHelpAccess := pHelpAccess^.pNext;
    end_while;
    pHelpAccess^.pNext$pVoid := ToStdLib.Malloc(size:=sizeof(t_AccessElement));
    pHelpAccess := pHelpAccess^.pNext;
  end_if;

  if pHelpAccess <> NIL then
    pHelpAccess^.eAccessType                  := AccessType;
    pHelpAccess^.usPlace                      := Place$USINT;
    pHelpAccess^.hiOffset                     := Offset;
    pHelpAccess^.uiLength                     := Length;
    pHelpAccess^.ppData                       := ppData;
    pHelpAccess^.ppStateByte                  := ppStateByte$^t_SDIAS_pStateByte;
    pHelpAccess^.ppControlByte                := ppControlByte$^t_SDIAS_pControlByte;
    pHelpAccess^.pWaitForAccess               := WaitForAccessHandle$^t_AccessElement;
    pHelpAccess^.udOSDOHandle                 := NIL;
    pHelpAccess^.pNext                        := NIL;
    pHelpAccess^.bCtrlAcc0                    := bCtrlAcc0;

    // count the data for the varan payload frames
    case AccessType of
      _Read:
          ISOWriteDO.Length += sizeof(t_SDIAS_ControlByte); // control byte
          ISOReadDO.Length  += sizeof(t_SDIAS_StateByte) + Length; // state byte + data length

      _Write:
          ISOWriteDO.Length += sizeof(t_SDIAS_ControlByte) + Length; // control byte + data length
          ISOReadDO.Length  += sizeof(t_SDIAS_StateByte); // state byte;

      _ReadDynamic:
          ISOWriteDO.Length += sizeof(t_SDIAS_ControlStructDynamic); // control byte + length info + offset info
          ISOReadDO.Length  += sizeof(t_SDIAS_StateByte) + Length; // state byte + data length

      _WriteDynamic:
          ISOWriteDO.Length += sizeof(t_SDIAS_ControlStructDynamic) + Length; // control byte + length info + offset info + data length
          ISOReadDO.Length  += sizeof(t_SDIAS_StateByte); // state byte;
    end_case;

    // only for easier debugging
    ModuleObjInfo[Place].AccessNo += 1;

    if pAccessHandle then
      pAccessHandle^ := pHelpAccess$UDINT;
    end_if;

    Success := TRUE;
  else
    ClassState := _MemoryFault;
    InitError := _MemoryFault;
    LogError("(SdiasManager::AddAccessToList) Failed to allocate memory for an SDIAS Access");

    if pAccessHandle then
      pAccessHandle^ := 0;
    end_if;

    Success := FALSE;
  end_if;

END_FUNCTION

FUNCTION VIRTUAL SdiasManager::ReceiveSDOResponse
	VAR_INPUT
		Command 	: t_SDIAS_SDO_Cmd;
		Offset 	: HINT;
		Length 	: USINT;
		Result 	: iprStates;
		pResponseBuffer 	: ^USINT;
		ResponseLength 	: USINT;
	END_VAR
	VAR_OUTPUT
		ret_code 	: iprStates;
	END_VAR

  ret_code := READY;

  case Command of
    SDIAS_SDO_CMD_REBUILD_SDIAS:
      // if it succeeded, check if we have something to do
      if Result = READY then
        // everthing is fine
      else
        // an error occured while performing the operation
        LogError("(SdiasManager::ReceiveSDOResponse) Rebuild SDIAS SDO command failed!");
      end_if;
    SDIAS_SDO_CMD_SET_NEW_END:
      // if it succeeded, check if we have something to do
      if Result = READY then
        // everthing is fine
        bReceivedNewEndRsp := TRUE;
      else
        // an error occured while performing the operation
        LogError("(SdiasManager::ReceiveSDOResponse) Set new DOL end command failed!");
      end_if;

  else
    ret_code := ERROR;
    LogError("(SdiasManager::ReceiveSDOResponse) Invalid command in SDO response!");
  end_case;

END_FUNCTION

FUNCTION SdiasManager::AddSDOReq
	VAR_INPUT
		pCmdSvr 	: ^SvrChCmd;
		Command 	: t_SDIAS_SDO_Cmd;
		Place 	: USINT;
		CmdLength 	: USINT;
		pReqBuf 	: ^USINT;
	END_VAR
	VAR_OUTPUT
		sd_retval 	: DINT;
	END_VAR

  // protect via mutex because this can be called from different task priorities
  OS_MT_WAIT(pv_Mutex);

  // if the buffer is full, or the next element in the buffer is already in use
  if (SDOHandling.pWrite^.Command <> SDIAS_SDO_CMD_INVALID) then
    sd_retval := SDIAS_MAILBOX_FULL;
    OS_MT_SIGNAL(pv_Mutex);
    return;
  end_if;

  // check the pointer first (if needed)
  if CmdLength then
    if pReqBuf then
      _memcpy(ptr1:=#SDOHandling.pWrite^.ReqBufData, ptr2:=pReqBuf, cntr:=CmdLength);
    else
      sd_retval := SDIAS_INVALID_PARAM_DATA_BUFFER;
      OS_MT_SIGNAL(pv_Mutex);
      return;
    end_if;
  end_if;

  SDOHandling.pWrite^.pCallBackSvr := pCmdSvr;
  SDOHandling.pWrite^.NMTCommand := 0;
  SDOHandling.pWrite^.SDIASPlace := Place;
  SDOHandling.pWrite^.CmdLength := CmdLength;

  case Command of
    SDIAS_SDO_CMD_MEM_READ,
    SDIAS_SDO_CMD_MEM_WRITE,
    SDIAS_SDO_CMD_CTRL_READ,
    SDIAS_SDO_CMD_CTRL_WRITE:
//    SDIAS_SDO_CMD_SPI_READ,
//    SDIAS_SDO_CMD_SPI_WRITE:
      // store offset and length for read and write accesses
      SDOHandling.pWrite^.RdWrHead := pReqBuf^$t_SDIAS_SDO_RdWr_Head;
    SDIAS_SDO_CMD_SPI_READ,
    SDIAS_SDO_CMD_SPI_WRITE:

      // store offset and length for read and write accesses
      SDOHandling.pWrite^.RdWrHead := pReqBuf^$t_SDIAS_SDO_RdWr_Head;

  end_case;

  // command is the last thing to store, because it indicates a complete entry
  SDOHandling.pWrite^.Command := Command;

  // we increment our used entries in the buffer (only for debugging)
  SDOHandling.EntriesUsed     += 1;

  // after we successfully added this SDO, set the write pointer to the next element
  if SDOHandling.pWrite = SDOHandling.pLastEntry then
    SDOHandling.pWrite := SDOHandling.pRingBufMemStart;
  else
    SDOHandling.pWrite += sizeof(t_SDORingBufEntry);
  end_if;

  sd_retval := SDIAS_OK;

  OS_MT_SIGNAL(pv_Mutex);

END_FUNCTION

FUNCTION SdiasManager::CyclicSDOHandling
  VAR
  	i,j           : USINT;
    FoundIt       : BOOL;
		Offset 	      : HINT;
		Length 	      : USINT;
    pTempChannel  : ^t_SDOChannel;
    TempChannel   : t_SDOChannel;
    pRingBufEntry : ^t_SDORingBufEntry;
    FirstFound    : USINT;
    LastFound     : USINT;
    Channels2Add  : DINT;
    StartIndex    : USINT;
    EndIndex      : USINT;
    pCmdSvr       : ^SvrChCmd;
  	tempCmd       : CmdStruct;
    _result       : results;
    ReceiveBuffer : ARRAY [0..127] OF USINT;
    ReceiveLength : UDINT;
    sd_retval     : DINT;
    TempUDINT     : UDINT;
    OldChannelNo  : USINT;
  END_VAR

  // protect via mutex because this can be called from different task priorities
  OS_MT_WAIT(pv_Mutex);

  if ConnectionType = SDIAS_CON_VIA_VARAN_uC then

    // check sdo response first. if a channel is ready it can be used for the next request

    // GET SDO RESPONSE
    if (AsyReadUsage = _NotUsed) | (AsyReadUsage = _UsedBySDO) then

      // if the AsyRdDO is used for polling, we check if we got a response
      if AsyReadUsage = _UsedBySDO then
        StartIndex := ((ASYReadDO.Offset - SDOHandling.OffsetSDOResp) / sizeof(t_SDOChannel))$USINT;
        EndIndex := StartIndex + (ASYReadDO.Length / sizeof(t_SDOChannel))$USINT - 1;
        Offset := 0;
        for i := StartIndex to EndIndex do
          if SDOHandling.aChannelData[i].WaitForResponse then
            // check for the response (copy only header first)
            _memcpy(ptr1:=#TempChannel, ptr2:=ASYReadDO.pData$^t_SDOChannel + Offset, cntr:=sizeof(t_SDOChannel) - sizeof(t_SDOChannel.Data));
            pRingBufEntry := SDOHandling.aChannelData[i].pActElement;

            // if the header info is mirrored, the SDO is ready
            if ((TempChannel.MessageCounter AND SDIAS_MASK_MESSAGE_COUNTER) = pRingBufEntry^.MessageCounter) &
               (TempChannel.SDIASPlace = pRingBufEntry^.SDIASPlace) &
               (TempChannel.Command$t_SDIAS_SDO_Cmd = pRingBufEntry^.Command) then

              // we got our response
              SDOHandling.aChannelData[i].WaitForResponse := FALSE;
              SDOHandling.EntriesUsed -= 1;

              // check for error
              if (TempChannel.MessageCounter AND SDIAS_MASK_GLOBAL_ERROR_FLAG) then
                tempCmd.aPara[3] := ERROR;
                // copy error info
                _memcpy(ptr1:=#TempChannel.Data, ptr2:=ASYReadDO.pData + t_SDOChannel.Data + Offset, cntr:=TempChannel.LengthOfData);

                // show error info
                case TempChannel.Data$DINT of
                  SDIAS_SDO_ERROR_INVALID_MSG_CNT:
                    LogValue("(SdiasManager::CyclicSDOHandling) SDO Error 0x{0}: Invalid message counter", TempChannel.Data$UDINT);

                  SDIAS_SDO_ERROR_MSG_CNT_NOT_SUCCESSIVE:
                    LogValue("(SdiasManager::CyclicSDOHandling) SDO Error 0x{0}: Message counter not successive", TempChannel.Data$UDINT);

                  SDIAS_SDO_ERROR_INVALID_CMD:
                    LogValue("(SdiasManager::CyclicSDOHandling) SDO Error 0x{0}: Invalid command", TempChannel.Data$UDINT);

                  SDIAS_SDO_ERROR_INVALID_SUBCMD:
                    LogValue("(SdiasManager::CyclicSDOHandling) SDO Error 0x{0}: Invalid subcommand", TempChannel.Data$UDINT);

                  SDIAS_SDO_ERROR_INVALID_PLACE:
                    LogValue("(SdiasManager::CyclicSDOHandling) SDO Error 0x{0}: Invalid SDIAS Place", TempChannel.Data$UDINT);

                  SDIAS_SDO_ERROR_INVALID_CMD_LENGTH:
                    LogValue("(SdiasManager::CyclicSDOHandling) SDO Error 0x{0}: Invalid length of data bytes", TempChannel.Data$UDINT);

                  SDIAS_SDO_ERROR_INVALID_ACCESS_OFFSET:
                    LogValue("(SdiasManager::CyclicSDOHandling) SDO Error 0x{0}: Invalid offset for access", TempChannel.Data$UDINT);

                  SDIAS_SDO_ERROR_INVALID_ACCESS_LENGTH:
                    LogValue("(SdiasManager::CyclicSDOHandling) SDO Error 0x{0}: Invalid length for access", TempChannel.Data$UDINT);

                  SDIAS_SDO_ERROR_INTERNAL_TIMEOUT:
                    LogValue("(SdiasManager::CyclicSDOHandling) SDO Error 0x{0}: Internal timeout", TempChannel.Data$UDINT);

                  SDIAS_SDO_ERROR_GENERAL_ERROR:
                    LogValue("(SdiasManager::CyclicSDOHandling) SDO Error 0x{0}: General Error", TempChannel.Data$UDINT);

                  SDIAS_SDO_ERROR_MSG_CNT_CHANGED:
                    LogValue("(SdiasManager::CyclicSDOHandling) SDO Error 0x{0}: Message counter changed while SDO request was processed", TempChannel.Data$UDINT);

                  SDIAS_SDO_ERROR_CLIENT_NOT_READY:
                    LogValue("(SdiasManager::CyclicSDOHandling) SDO Error 0x{0}: Communication error between SDIAS Manager and SDIAS Client", TempChannel.Data$UDINT);

                  SDIAS_SDO_ERROR_MNG_DPRAM_FAILURE:
                    LogValue("(SdiasManager::CyclicSDOHandling) SDO Error 0x{0}: Error accessing the SDIAS Manager DPRAM", TempChannel.Data$UDINT);

                  SDIAS_SDO_ERROR_ACCESS_NOT_ALLOWED:
                    LogValue("(SdiasManager::CyclicSDOHandling) SDO Error 0x{0}: Access not allowed (e.g. control access to SDIAS Manager)", TempChannel.Data$UDINT);

                  SDIAS_SDO_ERROR_FLASH_ACCESS_FAILED:
                    LogValue("(SdiasManager::CyclicSDOHandling) SDO Error 0x{0}: Flash access failed", TempChannel.Data$UDINT);

                  SDIAS_SDO_ERROR_INVALID_PARAMETERS:
                    LogValue("(SdiasManager::CyclicSDOHandling) SDO Error 0x{0}: Invalid parameters in SDO request", TempChannel.Data$UDINT);
                else
                  LogValue("(SdiasManager::CyclicSDOHandling) SDO Error 0x{0}: Unknown Error", TempChannel.Data$UDINT);
                end_case;
              else
                tempCmd.aPara[3]$iprStates := READY;
                // copy response data
                if TempChannel.LengthOfData then
                  if TempChannel.LengthOfData <= sizeof(t_SDOChannel.Data) then
                    _memcpy(ptr1:=#TempChannel.Data, ptr2:=ASYReadDO.pData + t_SDOChannel.Data + Offset, cntr:=TempChannel.LengthOfData);
                  else
                    LogValue("(SdiasManager::CyclicSDOHandling) SDO Error: Length in response is too big (0x{0} Byte; Max: 0x{1} Byte)", TempChannel.LengthOfData, sizeof(t_SDOChannel.Data));
                  end_if;
                end_if;
              end_if;

              // if there is a response, distribute it and set this channel to "available for the next SDO" (set command to SDIAS_SDO_CMD_INVALID and pChannel to NIL)
              tempCmd.uiCmd := SDIAS_CMD_SDO_RESPONSE;
              tempCmd.aPara[0] := TempChannel.Command$t_SDIAS_SDO_Cmd;

              // if we got response data
              if TempChannel.LengthOfData then

                // if the SDO command was successful
                if tempCmd.aPara[3]$iprStates = READY then

                  // check if it's a command with offset and length info
                  case TempChannel.Command$t_SDIAS_SDO_Cmd of
                    SDIAS_SDO_CMD_MEM_READ,
                    SDIAS_SDO_CMD_MEM_WRITE,
                    SDIAS_SDO_CMD_CTRL_READ,
                    SDIAS_SDO_CMD_CTRL_WRITE:
                      // save header info in extra parameters
                      tempCmd.aPara[1] := pRingBufEntry^.RdWrHead.Offset;
                      tempCmd.aPara[2] := pRingBufEntry^.RdWrHead.Length;

                      // remove header info for user from payload
                      TempChannel.LengthOfData -= sizeof(t_SDIAS_SDO_RdWr_Head);

                      // pointer to data
                      tempCmd.aPara[4] := (#TempChannel.Data + sizeof(t_SDIAS_SDO_RdWr_Head))$DINT;

                    SDIAS_SDO_CMD_SPI_READ,
                    SDIAS_SDO_CMD_SPI_WRITE:

                      // no length or offset available
                      tempCmd.aPara[1] := 0;
                      tempCmd.aPara[2] := 0;

                      // pointer to data
                      tempCmd.aPara[4] := (#TempChannel.Data)$DINT;

                  else
                      // no length or offset available
                      tempCmd.aPara[1] := 0;
                      tempCmd.aPara[2] := 0;

                      // pointer to data
                      tempCmd.aPara[4] := (#TempChannel.Data)$DINT;
                  end_case;
                else
                  // check if it's a command with offset and length info
                  case TempChannel.Command$t_SDIAS_SDO_Cmd of
                    SDIAS_SDO_CMD_MEM_READ,
                    SDIAS_SDO_CMD_MEM_WRITE,
                    SDIAS_SDO_CMD_CTRL_READ,
                    SDIAS_SDO_CMD_CTRL_WRITE,
                    SDIAS_SDO_CMD_SPI_READ,
                    SDIAS_SDO_CMD_SPI_WRITE:
                      // save header info in extra parameters
                      tempCmd.aPara[1] := pRingBufEntry^.RdWrHead.Offset;
                      tempCmd.aPara[2] := pRingBufEntry^.RdWrHead.Length;
                  end_case;

                  // pointer to error code
                  tempCmd.aPara[4] := (#TempChannel.Data)$DINT;
                end_if;
              else
                tempCmd.aPara[4] := 0;
              end_if;
              tempCmd.aPara[5] := TempChannel.LengthOfData;

              pCmdSvr := pRingBufEntry^.pCallBackSvr;

              if pCmdSvr$pVirtualBase^.NewInst(#tempCmd, #_result) <> READY then
                LogValue("(SdiasManager::CyclicSDOHandling) SDO Error: Error of module at place 0x{0} while receiving the SDO reponse (which was an ErrorCode)", i);
              end_if;

              // the position in the ringbuffer is free again
              pRingBufEntry^.BusyChannelNo := 0;
              pRingBufEntry^.Command := SDIAS_SDO_CMD_INVALID;

              // the SDO channel on the module is free again
              SDOHandling.aChannelData[i].pActElement := NIL;

            elsif (ops.tAbsolute - SDOHandling.aChannelData[i].RequestTime) >= SDIAS_SDO_TIMEOUT then
              // the SDO request timed out (should not happen)
              LogValue("(SdiasManager::CyclicSDOHandling) SDO Error: Timeout while waiting for answer of the SDIAS Manager µC (Channel {0} of range 1-3)", i+1);

              // we got our response
              SDOHandling.aChannelData[i].WaitForResponse := FALSE;
              SDOHandling.EntriesUsed -= 1;

              // distribute timeout error and set this channel to "available for the next SDO" (set command to SDIAS_SDO_CMD_INVALID and pChannel to NIL)
              tempCmd.uiCmd := SDIAS_CMD_SDO_RESPONSE;
              tempCmd.aPara[0] := pRingBufEntry^.Command$UINT;

              // check if it's a command with offset and length info
              case pRingBufEntry^.Command of
                SDIAS_SDO_CMD_MEM_READ,
                SDIAS_SDO_CMD_MEM_WRITE,
                SDIAS_SDO_CMD_CTRL_READ,
                SDIAS_SDO_CMD_CTRL_WRITE,
                SDIAS_SDO_CMD_SPI_READ,
                SDIAS_SDO_CMD_SPI_WRITE:
                  // save header info in extra parameters
                  tempCmd.aPara[1] := pRingBufEntry^.RdWrHead.Offset;
                  tempCmd.aPara[2] := pRingBufEntry^.RdWrHead.Length;
              else
                  // no length or offset available
                  tempCmd.aPara[1] := 0;
                  tempCmd.aPara[2] := 0;
              end_case;

              tempCmd.aPara[3] := ERROR;
              tempCmd.aPara[4] := 0;
              tempCmd.aPara[5] := 0; // no data available

              pCmdSvr := pRingBufEntry^.pCallBackSvr;
              if pCmdSvr$pVirtualBase^.NewInst(#tempCmd, #_result) <> READY then
                LogValue("(SdiasManager::CyclicSDOHandling) SDO Error: Error of module at place 0x{0} while receiving the SDO reponse", i);
              end_if;

              // the position in the ringbuffer is free again
              pRingBufEntry^.BusyChannelNo := 0;
              pRingBufEntry^.Command := SDIAS_SDO_CMD_INVALID;

              // the SDO channel on the module is free again
              SDOHandling.aChannelData[i].pActElement := NIL;
            end_if;
          end_if;

          Offset += sizeof(t_SDOChannel);
        end_for;
      end_if;

      // check for the first (needed for offset) and last (needed for length)
      Length := 0;
      FoundIt := FALSE;
      for i := 0 to (SDIAS_SDO_CHANNEL_NO-1) do
        if SDOHandling.aChannelData[i].pActElement & SDOHandling.aChannelData[i].WaitForResponse then
          if FoundIt = FALSE then
            // found first used channel
            FoundIt := TRUE;
            Offset := SDOHandling.OffsetSDOResp + i * sizeof(t_SDOChannel);
          end_if;
          Length += sizeof(t_SDOChannel);
        end_if;
      end_for;

      if FoundIt then

        // if we have pending SDO requests, start the AsyRdDO for polling
        if ChangeAsyRd(Offset:=Offset,
                       Length:=Length,
                       RunState:=_BUS_IF_RUN_STATE_CONT_RUN,
                       UsageType:=_UsedBySDO) = FALSE then
          LogError("(SdiasManager::CyclicSDOHandling) Error occured at starting the ReadDO for SDO polling");
        end_if;
      else
        // if all pending SDOs received stop DO
        if AsyReadUsage = _UsedBySDO then
          if ChangeAsyRd(Offset:=0,
                         Length:=0,
                         RunState:=_BUS_IF_RUN_STATE_NO_RUN,
                         UsageType:=_UsedBySDO) = FALSE then
            LogError("(SdiasManager::CyclicSDOHandling) Error occured at stopping the ReadDO");
          end_if;
        end_if;
      end_if;
    end_if;

    // SEND SDO REQUEST
    if (AsyWriteUsage = _NotUsed) | (AsyWriteUsage = _UsedBySDO) then
      // if there is a free channel on the module, we have unsent requests and the AsyWrDO is not used => send the Request (or more than 1 if possible)

      // first check if we need to increment the msg counter for a previously sent SDO message
      if SDOHandling.IncrementMsgCnt then
        for i := 0 to (SDIAS_SDO_CHANNEL_NO-1) do
          if SDOHandling.IncrementMsgCnt AND 1 then
            // next message counter for this channel
            if SDOHandling.aChannelData[i].MessageCnt = SDIAS_MASK_MESSAGE_COUNTER then
              SDOHandling.aChannelData[i].MessageCnt    := 0;
            else
              SDOHandling.aChannelData[i].MessageCnt    += 1;
            end_if;

            SDOHandling.aChannelData[i].pActElement^.MessageCounter := SDOHandling.aChannelData[i].MessageCnt;
            pTempChannel := #SDOHandling.aChannelData[i].ChannelData;
            pTempChannel^.MessageCounter  := SDOHandling.aChannelData[i].MessageCnt;

            // save the new message counter to the Varan DO
            _memcpy(ptr1:=ASYWriteDO.pData$^USINT + i * sizeof(t_SDOChannel) - (ASYWriteDO.Offset - SDOHandling.OffsetSDOReq)$USINT, ptr2:=pTempChannel, cntr:=pTempChannel^.LengthOfData + sizeof(t_SDOChannel) - sizeof(t_SDOChannel.Data));
            SDOHandling.aChannelData[i].WaitForResponse := TRUE;
            TempUDINT := ops.tAbsolute;
            SDOHandling.aChannelData[i].RequestTime     := TempUDINT;
          end_if;
          SDOHandling.IncrementMsgCnt := SDOHandling.IncrementMsgCnt SHR 1;
        end_for;

        // use the same length and offset (it's the same frame just with different message counters)
        Offset := ASYWriteDO.Offset;
        Length := ASYWriteDO.Length$USINT;

        // write the same frame again with higher message counter on the modified SDOs
        if ChangeAsyWr(Offset:=Offset,
                       Length:=Length,
                       RunState:=_BUS_IF_RUN_STATE_CONT_RUN,
                       UsageType:=_UsedBySDO) = FALSE then
          LogError("(SdiasManager::CyclicSDOHandling) Error occured at starting the WriteDO to write the new message counter");
        end_if;
      else
        // check for a free channel
        FoundIt := FALSE;
        for i := 0 to (SDIAS_SDO_CHANNEL_NO-1) do
          if SDOHandling.aChannelData[i].pActElement = NIL then
            // found a free channel
            FoundIt := TRUE;
            FirstFound := LastFound := i;
            Offset := SDOHandling.OffsetSDOReq + i * sizeof(t_SDOChannel);
            exit;
          end_if;
        end_for;

        // now we fill the buffer in the channels of the hardware (continue as long as there is space in the buffer and we have SDOs to send)
        Channels2Add := 0;
        while FoundIt & (SDOHandling.pRead^.Command <> SDIAS_SDO_CMD_INVALID) & (SDOHandling.pRead^.BusyChannelNo = 0) do
          // i is the index of the free channel => add the data
          pTempChannel := #SDOHandling.aChannelData[i].ChannelData;
          SDOHandling.aChannelData[i].pActElement     := SDOHandling.pRead;
          SDOHandling.pRead^.MessageCounter           := SDOHandling.aChannelData[i].MessageCnt;
          pTempChannel^.MessageCounter                := SDOHandling.pRead^.MessageCounter;
          pTempChannel^.NMT                           := SDOHandling.pRead^.NMTCommand;
          pTempChannel^.SDIASPlace                    := SDOHandling.pRead^.SDIASPlace;
          pTempChannel^.Command$t_SDIAS_SDO_Cmd       := SDOHandling.pRead^.Command;
          pTempChannel^.LengthOfData                  := SDOHandling.pRead^.CmdLength;
          if pTempChannel^.LengthOfData then
            _memcpy(ptr1:=#pTempChannel^.Data, ptr2:=#SDOHandling.pRead^.ReqBufData, cntr:=pTempChannel^.LengthOfData);
          end_if;

          // put the SDO request into the DPRAM on the right channel
          _memcpy(ptr1:=ASYWriteDO.pData$^t_SDOChannel + Channels2Add * sizeof(t_SDOChannel), ptr2:=pTempChannel, cntr:=pTempChannel^.LengthOfData + sizeof(t_SDOChannel) - sizeof(t_SDOChannel.Data));

          // remember this as the last found SDO to work with
          LastFound := i;

          // remember that we have to increment the message counter here
          SDOHandling.IncrementMsgCnt := SDOHandling.IncrementMsgCnt OR (1 SHL i);

          // this element is done by channel x
          SDOHandling.pRead^.BusyChannelNo := i+1;

          // increase channels to add
          Channels2Add += 1;

          // after we successfully added this SDO, set the read pointer to the next element
          if SDOHandling.pRead = SDOHandling.pLastEntry then
            SDOHandling.pRead := SDOHandling.pRingBufMemStart;
          else
            SDOHandling.pRead += sizeof(t_SDORingBufEntry);
          end_if;

          OldChannelNo := i;

          // check for a free channel
          FoundIt := FALSE;
          for i := 0 to (SDIAS_SDO_CHANNEL_NO-1) do
            if SDOHandling.aChannelData[i].pActElement = NIL then
              // found a free channel
              FoundIt := TRUE;

              if i > (OldChannelNo + 1) then
                // refresh the data in the DPRAM for the skipped channels
                for j := (OldChannelNo+1) to (i-1) do
                  // put the SDO request into the DPRAM on the right channel
                  _memcpy(ptr1:=ASYWriteDO.pData$^t_SDOChannel + j * sizeof(t_SDOChannel), ptr2:=#SDOHandling.aChannelData[j].ChannelData, cntr:=SDOHandling.aChannelData[j].ChannelData.LengthOfData + sizeof(t_SDOChannel) - sizeof(t_SDOChannel.Data));

                  // increase channels to add, because we also write the skipped ones
                  Channels2Add += 1;
                end_for;
              end_if;

              exit;
            end_if;
          end_for;
        end_while;

        if Channels2Add then
          Length := (LastFound - FirstFound + 1)$USINT * sizeof(t_SDOChannel);
          // if we have something to write => write it
          if ChangeAsyWr(Offset:=Offset,
                         Length:=Length,
                         RunState:=_BUS_IF_RUN_STATE_CONT_RUN,
                         UsageType:=_UsedBySDO) = FALSE then
            LogError("(SdiasManager::CyclicSDOHandling) Error occured at starting the WriteDO to write the new SDO command");
          end_if;
        elsif AsyWriteUsage = _UsedBySDO then
          // otherwise release the write buffer to other purposes
          if ChangeAsyWr(Offset:=0,
                         Length:=0,
                         RunState:=_BUS_IF_RUN_STATE_NO_RUN,
                         UsageType:=_UsedBySDO) = FALSE then
            LogError("(SdiasManager::CyclicSDOHandling) Error occured at stopping the WriteDO");
          end_if;
        end_if;
      end_if;
    end_if;
  else
    // if connected locally we can use the OS interfaces to access the SDO channels

    // check sdo response first. if a channel is ready it can be used for the next request

    // GET SDO RESPONSE
    if SDOHandling.EntriesUsed then
      // post init blocks the tasks in cyclic priority (the SDIAS Manager Code is running in lower priority than cyclic and has no time during the postinit) => give it some time
      if (b_PostInitFinished = FALSE) then
        ToMultiTask.TASKDELAY(timeout0:=SDIAS_WAIT_TIME_IN_POST_INIT);
      end_if;
      // check if we got a response
      for i := 0 to (SDIAS_SDO_CHANNEL_NO-1) do
        if SDOHandling.aChannelData[i].WaitForResponse then

          // get the SDO response
          ReceiveLength := 0;
          sd_retval := SDIAS_iReadSdoResponseChannel(udSdoHandle       := SDOHandling.aChannelData[i].SdoHandle
                                                   , udBufferLength    := sizeof(ReceiveBuffer)
                                                   , pucData           := #ReceiveBuffer[0]
                                                   , pudDataLength     := #ReceiveLength
                                                   );

          // check if it's finished => no more busy
          if sd_retval <> SDIAS_SDO_REQUEST_BUSY then
            if ReceiveLength <= sizeof(TempChannel.Data) then
              pRingBufEntry := SDOHandling.aChannelData[i].pActElement;

              // copy the info
              _memcpy(ptr1:= #TempChannel.Data, ptr2:= #ReceiveBuffer[0], cntr:= ReceiveLength);
              TempChannel.LengthOfData := ReceiveLength$USINT;
              TempChannel.Command$t_SDIAS_SDO_Cmd := pRingBufEntry^.Command;

              // we got our response
              SDOHandling.aChannelData[i].WaitForResponse := FALSE;
              SDOHandling.EntriesUsed -= 1;

              // check for error
              if sd_retval <> SDIAS_OK then
                tempCmd.aPara[3] := ERROR;

                LogSDOErrorInfo(sd_retval);
              else
                tempCmd.aPara[3]$iprStates := READY;
              end_if;

              // if there is a response, distribute it and set this channel to "available for the next SDO" (set command to SDIAS_SDO_CMD_INVALID and pChannel to NIL)
              tempCmd.uiCmd := SDIAS_CMD_SDO_RESPONSE;
              tempCmd.aPara[0] := pRingBufEntry^.Command$INT;

              // if we got response data
              if TempChannel.LengthOfData then

                // if the SDO command was successful
                if tempCmd.aPara[3]$iprStates = READY then

                  // check if it's a command with offset and length info
                  case TempChannel.Command$t_SDIAS_SDO_Cmd of
                    SDIAS_SDO_CMD_MEM_READ,
                    SDIAS_SDO_CMD_MEM_WRITE,
                    SDIAS_SDO_CMD_CTRL_READ,
                    SDIAS_SDO_CMD_CTRL_WRITE:
                      // save header info in extra parameters
                      tempCmd.aPara[1] := pRingBufEntry^.RdWrHead.Offset;
                      tempCmd.aPara[2] := pRingBufEntry^.RdWrHead.Length;

                      // remove header info for user from payload
                      TempChannel.LengthOfData -= sizeof(t_SDIAS_SDO_RdWr_Head);

                      // pointer to data
                      tempCmd.aPara[4] := (#TempChannel.Data + sizeof(t_SDIAS_SDO_RdWr_Head))$DINT;

                    SDIAS_SDO_CMD_SPI_READ,
                    SDIAS_SDO_CMD_SPI_WRITE:
                      // no length or offset available
                      tempCmd.aPara[1] := 0;
                      tempCmd.aPara[2] := 0;

                      // pointer to data
                      tempCmd.aPara[4] := (#TempChannel.Data)$DINT;

                  else
                      // no length or offset available
                      tempCmd.aPara[1] := 0;
                      tempCmd.aPara[2] := 0;

                      // pointer to data
                      tempCmd.aPara[4] := (#TempChannel.Data)$DINT;
                  end_case;
                else
                  // check if it's a command with offset and length info
                  case TempChannel.Command$t_SDIAS_SDO_Cmd of
                    SDIAS_SDO_CMD_MEM_READ,
                    SDIAS_SDO_CMD_MEM_WRITE,
                    SDIAS_SDO_CMD_CTRL_READ,
                    SDIAS_SDO_CMD_CTRL_WRITE,
                    SDIAS_SDO_CMD_SPI_READ,
                    SDIAS_SDO_CMD_SPI_WRITE:
                      // save header info in extra parameters
                      tempCmd.aPara[1] := pRingBufEntry^.RdWrHead.Offset;
                      tempCmd.aPara[2] := pRingBufEntry^.RdWrHead.Length;
                  end_case;

                  // pointer to error code
                  tempCmd.aPara[4] := (#sd_retval)$DINT;
                end_if;
              else
                tempCmd.aPara[4] := 0;
              end_if;
              tempCmd.aPara[5] := TempChannel.LengthOfData;

              pCmdSvr := pRingBufEntry^.pCallBackSvr;
              if pCmdSvr$pVirtualBase^.NewInst(#tempCmd, #_result) <> READY then
                LogValue("(SdiasManager::CyclicSDOHandling) SDO Error: Error of module at place 0x{0} while receiving the SDO reponse (which was an ErrorCode)", i);
              end_if;

              // the position in the ringbuffer is free again
              pRingBufEntry^.BusyChannelNo := 0;
              pRingBufEntry^.Command := SDIAS_SDO_CMD_INVALID;

              // the SDO channel on the module is free again
              SDOHandling.aChannelData[i].pActElement := NIL;
            else
              LogValue("(SdiasManager::CyclicSDOHandling) SDO Response too big. Received 0x{0} bytes. Maximum is 0x{1} bytes.", ReceiveLength, sizeof(TempChannel.Data));
            end_if;
          end_if;
        end_if;
      end_for;
    end_if;

    // SEND SDO REQUEST
    if SDOHandling.EntriesUsed then
      // if there is a free channel on the module and we have unsent requests => send the Requests

      // check for a free channel
      FoundIt := FALSE;
      for i := 0 to (SDIAS_SDO_CHANNEL_NO-1) do
        if SDOHandling.aChannelData[i].pActElement = NIL then
          // found a free channel
          FoundIt := TRUE;
          FirstFound := LastFound := i;
          exit;
        end_if;
      end_for;

      // now we fill the buffer in the channels of the hardware (continue as long as there is space in the buffer and we have SDOs to send)
      while FoundIt & (SDOHandling.pRead^.Command <> SDIAS_SDO_CMD_INVALID) & (SDOHandling.pRead^.BusyChannelNo = 0) do
        // i is the index of the free channel => add the data
        SDOHandling.aChannelData[i].pActElement     := SDOHandling.pRead;
        SDOHandling.pRead^.MessageCounter           := SDOHandling.aChannelData[i].MessageCnt;
        TempChannel.MessageCounter                  := SDOHandling.pRead^.MessageCounter;
        TempChannel.NMT                             := SDOHandling.pRead^.NMTCommand;
        TempChannel.SDIASPlace                      := SDOHandling.pRead^.SDIASPlace;
        TempChannel.Command$t_SDIAS_SDO_Cmd         := SDOHandling.pRead^.Command;
        TempChannel.LengthOfData                    := SDOHandling.pRead^.CmdLength;
        if TempChannel.LengthOfData then
          _memcpy(ptr1:=#TempChannel.Data, ptr2:=#SDOHandling.pRead^.ReqBufData, cntr:=TempChannel.LengthOfData);
        end_if;

        // send the SDO to the OS Interface
        sd_retval := SDIAS_iSendSdoRequestChannel(hManagerNodeHandle:= udNodeHandle
                                                , udChannel         := i
                                                , udCommand         := TempChannel.Command$t_SDIAS_SDO_Cmd
                                                , udSdiasAddress    := TempChannel.SDIASPlace
                                                , udDataLength      := TempChannel.LengthOfData
                                                , pucData           := #TempChannel.Data[0]
                                                , pudSdoHandle      := #SDOHandling.aChannelData[i].SdoHandle
                                                );

        if sd_retval = SDIAS_OK then
          // this element is done by channel x
          SDOHandling.pRead^.BusyChannelNo := i+1;

          SDOHandling.aChannelData[i].WaitForResponse := TRUE;
          TempUDINT := ops.tAbsolute;
          SDOHandling.aChannelData[i].RequestTime     := TempUDINT;

          // after we successfully added this SDO, set the read pointer to the next element
          if SDOHandling.pRead = SDOHandling.pLastEntry then
            SDOHandling.pRead := SDOHandling.pRingBufMemStart;
          else
            SDOHandling.pRead += sizeof(t_SDORingBufEntry);
          end_if;

          // check for a free channel
          FoundIt := FALSE;
          for i := 0 to (SDIAS_SDO_CHANNEL_NO-1) do
            if SDOHandling.aChannelData[i].pActElement = NIL then
              // found a free channel
              FoundIt := TRUE;
              exit;
            end_if;
          end_for;
        else
          LogSDOErrorInfo(sd_retval);
          exit;
        end_if;
      end_while;
    end_if;
  end_if;

    OS_MT_SIGNAL(pv_Mutex);

END_FUNCTION

FUNCTION SdiasManager::SetRequiredError
	VAR_INPUT
		pTargetThis 	: ^SdiasBase;(* := NIL *)
		Place 	: UDINT;(* := SDIAS_PLACE_NO_MODULE_ADDED_SO_FAR *)
	END_VAR
  VAR
  	tempCmd         : CmdStruct;
    _result         : results;
    i : UDINT;
    FoundIt : BOOL;
  END_VAR

  if pTargetThis & (Place <> SDIAS_PLACE_NO_MODULE_ADDED_SO_FAR) then
    pTargetThis^.ClassState := _RequiredError;

    LogValue("(SdiasManager::SetRequiredError) Required Error on SDIAS Place 0x{0}", Place);
  else
    // general required error (initialisation failed) => search for the first required module to blame (if there is one)
    FoundIt := FALSE;
    if MaxPlace <> SDIAS_PLACE_NO_MODULE_ADDED_SO_FAR then
      for i := 0 to MaxPlace do
        if ModuleObjInfo[i].pThis & ModuleObjInfo[i].Required then
          FoundIt := TRUE;
        end_if;
      end_for;
    end_if;

    // if no required module => don't crash
    if FoundIt = FALSE then
      return;
    end_if;
  end_if;

  ClassState := _RequiredError;

  // set required error
  tempCmd.uiCmd     := _BUS_IF_SET_REQUIRED_ERROR;

  ToBusInterface.NewInst(pPara:=#tempCmd, pResult:=#_result);
  if _result.aData[0]$t_BusIFRetvalErrorcode <> _BUS_IF_RETVAL_OK then
    LogError("(SdiasManager::SetRequiredError) Failed to set required error to BusInterface");
  end_if;

  if InitSSW <> _PrepareError then
    ErrorInitStep := InitSSW;
    InitSSW := _PrepareError;
  end_if;

END_FUNCTION

// New interface - 2013-05-28
// -----------------------------------------------------------------------
// -	bIsWriteAcc0 : 0 - read access , 1 - write access
// -	iModAddr0 : Module adress at sdias bus (device adr + offset)
// -	iDataLen0 : Data length
// -	bCtrlAcc0 : 0 - access to regular memory, 1 > access to ctrl access
// -    bAccList0 : 0 - access to iso read/write list, 1 - acc to manager admin list, 2 - access to sdo list, 3 - access to periodic manager list

FUNCTION SdiasManager::DOL_Handling_Add_DO_TO_List
	VAR_INPUT
		bIsWriteAcc0 	: UDINT;
		iModAddr0 	: HDINT;
		iDataLen0 	: UINT;
		bCtrlAcc0 	: UDINT;
		iWaitDOOffset0 	: UINT;
		bIsDynamic0 	: BOOL;
		pActAccess0 	: ^t_AccessElement;
	END_VAR
	VAR_OUTPUT
		iRetCode 	: DINT;
	END_VAR
  VAR
    pReadList       : ^t_SDIAS_DOL_DESC;
    pWriteList      : ^t_SDIAS_DOL_DESC;
    iEndDataPointRd : UINT;
    iEndDOLPointRd  : UDINT;
    iEndDataPointWr : UINT;
    iEndDOLPointWr  : UDINT;
    udCmdType       : UDINT;
    ReadLen         : UINT;
    ReadAdd         : HDINT;
    WriteLen        : UINT;
    WriteAdd        : HDINT;
    udDOFlags       : UDINT;
  END_VAR

  iRetCode := -1;

  (* Only ISO DOL	in hardware classes *)
  pReadList := #gcRead_DOL_Desc;
  pWriteList := #gcWrite_DOL_Desc;

  if ConnectionType = SDIAS_CON_VIA_VARAN_uC then

    (*	Check endpoints of data and DOL	*)
    iEndDataPointRd := pReadList^.iBaseAddrData + pReadList^.iOffLastData + 1;
    iEndDOLPointRd  := pReadList^.iBaseAddr + pReadList^.iOffEndCmd;

    iEndDataPointWr := pWriteList^.iBaseAddrData + pWriteList^.iOffLastData +  1;
    iEndDOLPointWr  := pWriteList^.iBaseAddr + pWriteList^.iOffEndCmd;

    if(bIsWriteAcc0 = 0) then
      (*	Check endpoints of data and DOL	*)
      iEndDataPointRd += iDataLen0;
      iEndDOLPointRd  += sizeof(t_SDIAS_STD_CMD_DO);
    else
      (*	Check endpoints of data and DOL	*)
      iEndDataPointWr += iDataLen0;
      iEndDOLPointWr  += sizeof(t_SDIAS_STD_CMD_DO);
    end_if;

    (* Check available data	in read space *)
    if(iEndDataPointRd > pReadList^.iEndAddrData) then
      iRetCode := -3;
    (* Check space in DOL	*)
    elsif(iEndDOLPointRd > pReadList^.iEndAddr) then
      iRetCode := -4;
    (* Check available data	in write space *)
    elsif(iEndDataPointWr > pWriteList^.iEndAddrData) then
      iRetCode := -5;
    (* Check space in DOL	*)
    elsif(iEndDOLPointWr > pWriteList^.iEndAddr) then
      iRetCode := -6;
    (* Space for all required data	*)
    else

      // Add 1 to switch to first empty byte
      pWriteList^.iOffLastData += sizeof(t_SDIAS_ControlByte);										(* Add do ctrl byte to data		*)
      pReadList^.iOffLastData += sizeof(t_SDIAS_StateByte);

      pWriteList^.iOffFirstData := pWriteList^.iOffLastData;			(* Store data start points		*)
      pReadList^.iOffFirstData := pReadList^.iOffLastData;

      // dynamic accesses need more bytes in the write payload
      if bIsDynamic0 then
        // control byte is already considered, so we have to add the difference here
        pWriteList^.iOffLastData += (sizeof(t_SDIAS_ControlStructDynamic) - sizeof(t_SDIAS_ControlByte));
      end_if;

      cModulAccessCmds[0].OffsetWritePayload := pWriteList^.iBaseAddrData + pWriteList^.iOffFirstData;		(* Store data offsets			*)
      cModulAccessCmds[0].OffsetReadPayload := pReadList^.iBaseAddrData + pReadList^.iOffFirstData;

      (* Set wait for DO to inactive	*)
      cModulAccessCmds[0].OffsetVolatileWaitFlag := iWaitDOOffset0;

      (* Init scratchpad info to 0	*)
      cModulAccessCmds[0].ErrorInfo := 0;

      (* Ctrl access *)
      if(bCtrlAcc0 <> 0) then
        (* Ctrl access +  retrys	*)
        cModulAccessCmds[0].CmdRetries  := SDIAS_CMD_ACC_CONTROL + (SDIAS_RETRIES_ALLOWED shl 5);
      else
        (* Mem access +  retrys	*)
        cModulAccessCmds[0].CmdRetries  := SDIAS_CMD_ACC_MEMORY + (SDIAS_RETRIES_ALLOWED shl 5);
      end_if;

      (* Init reserved info to 0	*)
      cModulAccessCmds[0].Reserved := 0;

      (* Write command to dpram 	*)
      if(bIsWriteAcc0 = 0) then

        cModulAccessCmds[0].ReadLength := to_usint(iDataLen0);
        cModulAccessCmds[0].ReadOffset := to_uint(iModAddr0);

        cModulAccessCmds[0].WriteLength := 0;
        cModulAccessCmds[0].WriteOffset  := 0;

        (* Store write adress of new command  *)
        uiWriteCmdAddr := pReadList^.iBaseAddr + pReadList^.iOffEndCmd;

        (* Increment offset of end command	*)
        pReadList^.iOffEndCmd += sizeof(t_SDIAS_STD_CMD_DO);

        (* End of list	*)
        DOL_Handling_Create_End_Cmd(#cModulAccessCmds[1]);

        (* Add read length to iso read usage	*)
        pReadList^.iOffLastData += iDataLen0;

        (* Set usage vars	*)
        pReadList^.iUsageData := pReadList^.iOffLastData + 1;
        pReadList^.iUsageDOL := pReadList^.iOffEndCmd + sizeof(t_SDIAS_STD_CMD_DO);

        pWriteList^.iUsageData := pWriteList^.iOffLastData + 1;

      else

        cModulAccessCmds[0].ReadLength := 0;
        cModulAccessCmds[0].ReadOffset := 0;

        cModulAccessCmds[0].WriteLength := to_usint(iDataLen0);
        cModulAccessCmds[0].WriteOffset  := to_uint(iModAddr0);

        (* Store write adress of new command  *)
        uiWriteCmdAddr := pWriteList^.iBaseAddr + pWriteList^.iOffEndCmd;

        (* Increment offset of end command	*)
        pWriteList^.iOffEndCmd += sizeof(t_SDIAS_STD_CMD_DO);

        (* End of list	*)
        DOL_Handling_Create_End_Cmd(#cModulAccessCmds[1]);

        (* Add write length to iso write usage	*)
        pWriteList^.iOffLastData += iDataLen0;

        (* Set usage vars	*)
        pReadList^.iUsageData := pReadList^.iOffLastData + 1;

        pWriteList^.iUsageData := pWriteList^.iOffLastData + 1;
        pWriteList^.iUsageDOL := pWriteList^.iOffEndCmd + sizeof(t_SDIAS_STD_CMD_DO);

        (* Reset write payload	*)
        //SDIAS_Module_CPLD_Com_Write_Data(pWriteList^.iBaseAddrData + pWriteList^.iOffFirstData + 1, iDataLen0 , (void *)&iDOL_ResetData[0]);

      end_if;

      iRetCode := 0;

    end_if;

  else
    // locally we use the OS interface to create the DO

    (* Ctrl access *)
    if(bCtrlAcc0 <> 0) then
      (* Ctrl access +  retrys	*)
      udCmdType         := SDIAS_CMD_ACC_CONTROL;
    else
      (* Mem access +  retrys	*)
      udCmdType         := SDIAS_CMD_ACC_MEMORY;
    end_if;

    // if the interface for dynamic DOs is not available => use the old interface
    if (pSDIAS^.udVersion < SDIAS_CIL_VERSION_SUPPORTS_DYNAMIC_DO) then
      iRetCode := SDIAS_iAddDo(hNodeHandle         := udNodeHandle
                             , udDolType           := SDIAS_DOL_TYPE_ISO
                             , udCmdType           := udCmdType
                             , udRetries           := SDIAS_RETRIES_ALLOWED
                             , udIsWriteAcc        := bIsWriteAcc0
                             , udModuleAddress     := iModAddr0
                             , udDataLen           := iDataLen0
                             , hAddrVolatileWait   := iWaitDOOffset0
                             , phAddrWriteData     := (#cModulAccessCmds[0].OffsetWritePayload)$^pVoid
                             , phAddrReadData      := (#cModulAccessCmds[0].OffsetReadPayload)$^pVoid
                             );
    else
      // make read and write settings
      if bIsWriteAcc0 then
        WriteLen := iDataLen0;
        WriteAdd := iModAddr0;
        ReadLen  := 0;
        ReadAdd  := 0;
      else
        WriteLen := 0;
        WriteAdd := 0;
        ReadLen  := iDataLen0;
        ReadAdd  := iModAddr0;
      end_if;

      // set DO flags
      if bIsDynamic0 then
        if bIsWriteAcc0 then
          udDOFlags := SDIAS_DO_FLAG_SUPPORT_VARIABLE_READ_BYTE_COUNT_AND_MODULE_ADDR;
        else
          udDOFlags := SDIAS_DO_FLAG_SUPPORT_VARIABLE_WRITE_BYTE_COUNT_AND_MODULE_ADDR;
        end_if;
      else
        udDOFlags := 0;
      end_if;

      // use the new interface
      iRetCode := SDIAS_iAddDoDynamic(hNodeHandle         := udNodeHandle
                                    , udDolType           := SDIAS_DOL_TYPE_ISO
                                    , udCmdType           := udCmdType
                                    , udSubCmdType        := SDIAS_DO_SUBCMD_NONE
                                    , udRetries           := SDIAS_RETRIES_ALLOWED
                                    , udReadAddress       := ReadAdd
                                    , udReadDataLen       := ReadLen
                                    , udWriteAddress      := WriteAdd
                                    , udWriteDataLen      := WriteLen
                                    , udAddrVolatileWait  := iWaitDOOffset0
                                    , hJumpDoHandle       := SDIAS_INVALID_VOLATILE_WAIT_HANDLE
                                    , udDoFlags           := udDOFlags
                                    , phDoHandle          := #pActAccess0^.udOSDOHandle
                                    , phAddrWriteData     := (#cModulAccessCmds[0].OffsetWritePayload)$^pVoid
                                    , phAddrReadData      := (#cModulAccessCmds[0].OffsetReadPayload)$^pVoid
                                    );
    end_if;

    if iRetCode = SDIAS_OK then
      (* Store data offsets			*)
      pWriteList^.iOffFirstData := cModulAccessCmds[0].OffsetWritePayload - pWriteList^.iBaseAddrData;
      pReadList^.iOffFirstData  := cModulAccessCmds[0].OffsetReadPayload  - pReadList^.iBaseAddrData;
    else
      LogError("(SdiasManager::DOL_Handling_Add_DO_TO_List) Failed to add custom SDIAS access via OS interface!");
    end_if;
  end_if;

END_FUNCTION

FUNCTION SdiasManager::DOL_Handling_Create_End_Cmd
	VAR_INPUT
		pEndCmdBuffer 	: ^t_SDIAS_DOListEntry;
	END_VAR

 	(* End of list	*)
	pEndCmdBuffer^.OffsetReadPayload := 0xFFFF;
	pEndCmdBuffer^.OffsetWritePayload := 0xFFFF;

	(* Set wait for DO to inactive	*)
	pEndCmdBuffer^.OffsetVolatileWaitFlag := SDIAS_INVALID_VOLATILE_WAIT_HANDLE;

	(* Init scratchpad info to 0	*)
	pEndCmdBuffer^.ErrorInfo := 0;

	pEndCmdBuffer^.CmdRetries := 0x0;

	pEndCmdBuffer^.ReadLength := 0;
	pEndCmdBuffer^.ReadOffset := 0;

	(* Init reserved info to 0	*)
	pEndCmdBuffer^.Reserved := 0;

	pEndCmdBuffer^.WriteLength := 0;
	pEndCmdBuffer^.WriteOffset  := 0;

END_FUNCTION

FUNCTION SdiasManager::LogSDOErrorInfo
	VAR_INPUT
		OSRetVal 	: DINT;
	END_VAR

 // show error info
  case OSRetVal of
    SDIAS_MAILBOX_FULL:
      LogValue("(SdiasManager::LogSDOErrorInfo) SDO Error 0x{0}: Mailbox full", (0-OSRetVal)$UDINT);

    SDIAS_TIMEOUT_TASK:
      LogValue("(SdiasManager::LogSDOErrorInfo) SDO Error 0x{0}: Timeout of task", (0-OSRetVal)$UDINT);

    SDIAS_RESPONSE_BUFFER_TOO_SMALL:
      LogValue("(SdiasManager::LogSDOErrorInfo) SDO Error 0x{0}: Response buffer too small", (0-OSRetVal)$UDINT);

    SDIAS_TIMEOUT_SDO_RESPONSE:
      LogValue("(SdiasManager::LogSDOErrorInfo) SDO Error 0x{0}: Timeout SDO response", (0-OSRetVal)$UDINT);

    SDIAS_OUT_OF_HANDLES:
      LogValue("(SdiasManager::LogSDOErrorInfo) SDO Error 0x{0}: Out of handles", (0-OSRetVal)$UDINT);

    SDIAS_INVALID_PARAM_DATA_LENGTH:
      LogValue("(SdiasManager::LogSDOErrorInfo) SDO Error 0x{0}: Invalid length of data bytes", (0-OSRetVal)$UDINT);

    SDIAS_INVALID_PARAM_DATA_BUFFER:
      LogValue("(SdiasManager::LogSDOErrorInfo) SDO Error 0x{0}: Invalid data buffer", (0-OSRetVal)$UDINT);

    SDIAS_INVALID_PARAM_SDO_HANDLE:
      LogValue("(SdiasManager::LogSDOErrorInfo) SDO Error 0x{0}: Invalid SDO handle", (0-OSRetVal)$UDINT);

    SDIAS_INVALID_PARAM_NODE:
      LogValue("(SdiasManager::LogSDOErrorInfo) SDO Error 0x{0}: Invalid node handle", (0-OSRetVal)$UDINT);

    SDIAS_GLOBAL_ERROR:
      LogValue("(SdiasManager::LogSDOErrorInfo) SDO Error 0x{0}: General Error of SDIAS Manager", (0-OSRetVal)$UDINT);

    SDIAS_INVALID_MANAGER:
      LogValue("(SdiasManager::LogSDOErrorInfo) SDO Error 0x{0}: SDIAS Manager not found", (0-OSRetVal)$UDINT);

    SDIAS_SENDING_SDO_REQUEST_FAILED:
      LogValue("(SdiasManager::LogSDOErrorInfo) SDO Error 0x{0}: Sending SDO request failed", (0-OSRetVal)$UDINT);

    SDIAS_RECEIVING_SDO_RESPONSE_FAILED:
      LogValue("(SdiasManager::LogSDOErrorInfo) SDO Error 0x{0}: Receiving SDO response failed", (0-OSRetVal)$UDINT);

    SDIAS_MANAGER_GLOBAL_ERROR:
      LogValue("(SdiasManager::LogSDOErrorInfo) SDO Error 0x{0}: General Error of SDIAS Manager (like communication problems to client)", (0-OSRetVal)$UDINT);

    SDIAS_INTERNAL_ERROR:
      LogValue("(SdiasManager::LogSDOErrorInfo) SDO Error 0x{0}: Internal error", (0-OSRetVal)$UDINT);
  else
    LogValue("(SdiasManager::LogSDOErrorInfo) SDO Error 0x{0}: Unknown Error", (0-OSRetVal)$UDINT);
  end_case;

END_FUNCTION

FUNCTION SdiasManager::CheckAccess
	VAR_INPUT
		bsStateByte 	: t_SDIAS_StateByte;
		sdRequired 	: DINT;
		sdPlace 	: DINT;
		pCrashThisTime 	: ^USINT;
		pCrashMessage 	: ^CHAR;
	END_VAR
	VAR_OUTPUT
		usRetryCounter 	: USINT;
	END_VAR

  // increase retrycounter if retries occured on the access
  usRetryCounter := bsStateByte SHR 5;

  // check if the access failed
  if sdRequired & (bsStateByte.AccessFailed = TRUE) then
    ModuleObjInfo[sdPlace].pThis^.ClassState := _RequiredError;
    RequiredPlace := sdPlace;
    CyclicMsgMarker.PostIt.RequiredError := TRUE;
    ClassState := _RequiredError;
    ErrorInitStep := InitSSW;
    InitSSW := _PrepareError;

    pCrashThisTime^ := 2;

    _strcpy(dest:=pCrashMessage, src:="Access to a required SDIAS Module failed");
  end_if;

END_FUNCTION

FUNCTION SdiasManager::PostRtMessages

  // if there are some messages to post, post them (the methods in the brackets are not the actual, but the methods were the error occured)
  if CyclicMsgMarker.PostIt then
    if CyclicMsgMarker.PostIt.IsoReadRunFailed then
      LogError("(SdiasManager::RtWork) Error changing the run state of the isochronous read access!");
    end_if;

    if CyclicMsgMarker.PostIt.IsoWriteRunFailed then
      LogError("(SdiasManager::RtWork) Error changing the run state of the isochronous write access!");
    end_if;

    if CyclicMsgMarker.PostIt.RequiredError then
      LogValue("(SdiasManager::RtWork) Required Error at SDIAS Place 0x{0}", RequiredPlace$UDINT);
    end_if;

    if CyclicMsgMarker.PostIt.ForwardRequiredErrorFailed then
      LogError("(SdiasManager::RtWork) Failed to set required error to BusInterface");
    end_if;

    if CyclicMsgMarker.PostIt.ToggleErrorWrTask & (CyclicMsgMarker.AlreadyPosted.ToggleErrorWrTask = FALSE) then
      LogError("(SdiasManager::RtWork) Error at toggle bit of iso write task of SDIAS");
      CyclicMsgMarker.AlreadyPosted.ToggleErrorWrTask := TRUE;
    end_if;

    if CyclicMsgMarker.PostIt.ToggleErrorRdTask & (CyclicMsgMarker.AlreadyPosted.ToggleErrorRdTask = FALSE) then
      LogError("(SdiasManager::RtWork) Error at toggle bit of iso read task of SDIAS");
      CyclicMsgMarker.AlreadyPosted.ToggleErrorRdTask := TRUE;
    end_if;

    if CyclicMsgMarker.PostIt.ErrorWrTask & (CyclicMsgMarker.AlreadyPosted.ErrorWrTask = FALSE) then
      LogValue("(SdiasManager::RtWork) Error at iso write task of SDIAS 0x{0}", (WriteTaskInfo.pReadData^.ErrorInfoFlags AND SDIAS_ERROR_INFO_MASK));
      CyclicMsgMarker.AlreadyPosted.ErrorWrTask := TRUE;
    end_if;

    if CyclicMsgMarker.PostIt.ErrorRdTask & (CyclicMsgMarker.AlreadyPosted.ErrorRdTask = FALSE) then
      LogValue("(SdiasManager::RtWork) Error at iso read task of SDIAS 0x{0}", (ReadTaskInfo.pReadData^.ErrorInfoFlags AND SDIAS_ERROR_INFO_MASK));
      CyclicMsgMarker.AlreadyPosted.ErrorRdTask := TRUE;
    end_if;

    if CyclicMsgMarker.PostIt.GetRdInfoFailed & (CyclicMsgMarker.AlreadyPosted.GetRdInfoFailed = FALSE) then
      LogError("(SdiasManager::RtWork) Error fetching iso read task info from OS");
      CyclicMsgMarker.AlreadyPosted.GetRdInfoFailed := TRUE;
    end_if;

    if CyclicMsgMarker.PostIt.GetWrInfoFailed & (CyclicMsgMarker.AlreadyPosted.GetWrInfoFailed = FALSE) then
      LogError("(SdiasManager::RtWork) Error fetching iso read task info from OS");
      CyclicMsgMarker.AlreadyPosted.GetWrInfoFailed := TRUE;
    end_if;

    if CyclicMsgMarker.PostIt.SetSyncFailed & (CyclicMsgMarker.AlreadyPosted.SetSyncFailed = FALSE) then
      LogError("(SdiasManager::RtWork) Failed to set sync out of pll");
      CyclicMsgMarker.AlreadyPosted.SetSyncFailed := TRUE;
    end_if;

    if CyclicMsgMarker.PostIt.GetFrameCounterFailed & (CyclicMsgMarker.AlreadyPosted.GetFrameCounterFailed = FALSE) then
      LogError("(SdiasManager::RtWork) Failed to get the frame counter info via OS interface");
      CyclicMsgMarker.AlreadyPosted.SetSyncFailed := TRUE;
    end_if;

    if CyclicMsgMarker.PostIt.WrTaskNotFinished & (CyclicMsgMarker.AlreadyPosted.WrTaskNotFinished = FALSE) then
      LogError("(SdiasManager::RtWork) Iso write task of SDIAS hasn't been completed");
      CyclicMsgMarker.AlreadyPosted.WrTaskNotFinished := TRUE;
    end_if;
